KUKA KRL program: MyProgram_261().src

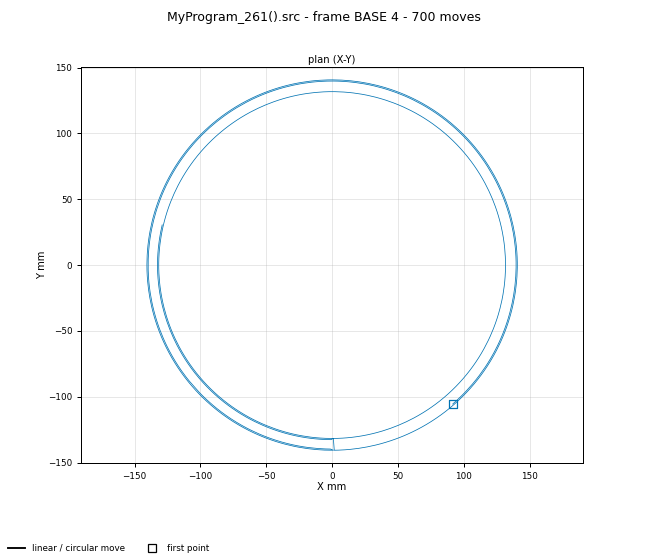
[picture p0: tool path of MyProgram_261().src in frame BASE 4, 700 of 700 moves have a stored position in this frame; points joined in program order, loops and branches not executed]
&ACCESS RVP
&REL 1
&PARAM TEMPLATE = C:\KRC\Roboter\Template\vorgabe
&PARAM EDITMASK = *
DEF MyProgram_261()
; ---- Setting reference (Base) ----
$BASE = BASE_DATA[4]

; --------------------------
; ---- Setting tool (TCP) ----
$TOOL = TOOL_DATA[3]
; --------------------------

$VEL.CP = VEL_APROX_PRINT
Startdeposition()
$VEL.CP = VEL_PRINT
LIN {X 91.5641,Y -105.5232,Z 167,A -46.4819,B 10.3454,C 0.2942,E1 10.4568,E2 497.4556} C_DIS
LIN {X 94.9436,Y -102.4931,Z 167,A -45.04,B 10.3452,C 0.3012,E1 10.4597,E2 496.067} C_DIS
LIN {X 98.56,Y -99.0198,Z 167,A -43.0358,B 10.3452,C 0.2981,E1 10.4637,E2 494.0674} C_DIS
LIN {X 101.6375,Y -95.8582,Z 167,A -40.8516,B 10.3456,C 0.2845,E1 10.468,E2 491.8321} C_DIS
LIN {X 104.5658,Y -92.6553,Z 167,A -39.6802,B 10.3453,C 0.2962,E1 10.47,E2 490.7387} C_DIS
LIN {X 106.6015,Y -90.306,Z 167,A -38.2518,B 10.3455,C 0.2893,E1 10.4727,E2 489.2889} C_DIS
LIN {X 109.2383,Y -87.0977,Z 167,A -36.5625,B 10.3456,C 0.2857,E1 10.4756,E2 487.5994} C_DIS
LIN {X 111.7975,Y -83.7884,Z 167,A -34.7726,B 10.3458,C 0.2796,E1 10.4787,E2 485.798} C_DIS
LIN {X 116.3977,Y -77.2703,Z 167,A -31.7918,B 10.3458,C 0.2792,E1 10.4834,E2 482.8518} C_DIS
LIN {X 118.3157,Y -74.3,Z 167,A -29.8592,B 10.3462,C 0.2629,E1 10.4864,E2 480.8544} C_DIS
LIN {X 120.3509,Y -70.9556,Z 167,A -28.8973,B 10.3459,C 0.2756,E1 10.4876,E2 479.975} C_DIS
LIN {X 122.8521,Y -66.5321,Z 167,A -26.472,B 10.3463,C 0.2612,E1 10.491,E2 477.5029} C_DIS
LIN {X 125.5362,Y -61.3138,Z 167,A -24.2471,B 10.3463,C 0.2596,E1 10.4938,E2 475.299} C_DIS
LIN {X 126.9956,Y -58.2302,Z 167,A -22.8435,B 10.3463,C 0.2557,E1 10.4954,E2 473.8932} C_DIS
LIN {X 128.5472,Y -54.7236,Z 167,A -21.1883,B 10.3465,C 0.2492,E1 10.4973,E2 472.2256} C_DIS
LIN {X 129.9617,Y -51.2729,Z 167,A -19.845,B 10.3465,C 0.2499,E1 10.4986,E2 470.9048} C_DIS
LIN {X 131.4593,Y -47.2962,Z 167,A -17.9921,B 10.3467,C 0.2421,E1 10.5004,E2 469.0356} C_DIS
LIN {X 132.6867,Y -43.7365,Z 167,A -16.549,B 10.3467,C 0.2405,E1 10.5017,E2 467.6039} C_DIS
LIN {X 133.7753,Y -40.2869,Z 167,A -14.9397,B 10.3469,C 0.233,E1 10.503,E2 465.9767} C_DIS
LIN {X 134.9483,Y -36.159,Z 167,A -12.8239,B 10.3472,C 0.2185,E1 10.5046,E2 463.8124} C_DIS
LIN {X 136.0946,Y -31.5754,Z 167,A -11.579,B 10.347,C 0.2313,E1 10.5054,E2 462.6559} C_DIS
LIN {X 136.6271,Y -29.183,Z 167,A -10.1588,B 10.3473,C 0.2174,E1 10.5062,E2 461.1805} C_DIS
LIN {X 137.2908,Y -25.8822,Z 167,A -9.1019,B 10.3472,C 0.222,E1 10.5068,E2 460.1643} C_DIS
LIN {X 137.8805,Y -22.5325,Z 167,A -7.7697,B 10.3472,C 0.2196,E1 10.5074,E2 458.8388} C_DIS
LIN {X 138.4173,Y -18.9686,Z 167,A -6.2808,B 10.3473,C 0.215,E1 10.508,E2 457.347} C_DIS
LIN {X 138.8085,Y -15.8511,Z 167,A -4.951,B 10.3474,C 0.2102,E1 10.5084,E2 456.0104} C_DIS
LIN {X 139.2347,Y -11.5036,Z 167,A -3.2691,B 10.3474,C 0.2078,E1 10.5089,E2 454.3408} C_DIS
LIN {X 139.4553,Y -8.4152,Z 167,A -1.8781,B 10.3476,C 0.2009,E1 10.5091,E2 452.9329} C_DIS
LIN {X 139.6307,Y -4.7299,Z 167,A -0.5083,B 10.3476,C 0.2003,E1 10.5093,E2 451.5801} C_DIS
LIN {X 139.698,Y -1.8215,Z 167,A 0.7879,B 10.3477,C 0.194,E1 10.5093,E2 450.2693} C_DIS
LIN {X 139.6853,Y 2.585,Z 167,A 2.554,B 10.3477,C 0.1898,E1 10.5093,E2 448.5067} C_DIS
LIN {X 139.5635,Y 6.4013,Z 167,A 4.1323,B 10.3479,C 0.1849,E1 10.5091,E2 446.9253} C_DIS
LIN {X 139.2836,Y 10.9175,Z 167,A 5.8225,B 10.3479,C 0.1839,E1 10.5088,E2 445.2548} C_DIS
LIN {X 138.9636,Y 14.4206,Z 167,A 7.4324,B 10.348,C 0.1753,E1 10.5083,E2 443.6218} C_DIS
LIN {X 138.2126,Y 20.4014,Z 167,A 9.8969,B 10.3482,C 0.1683,E1 10.5074,E2 441.156} C_DIS
LIN {X 137.4569,Y 24.9855,Z 167,A 11.6074,B 10.3482,C 0.168,E1 10.5066,E2 439.4689} C_DIS
LIN {X 136.0935,Y 31.5801,Z 167,A 14.2954,B 10.3482,C 0.1621,E1 10.505,E2 436.7881} C_DIS
LIN {X 135.3473,Y 34.6364,Z 167,A 15.6039,B 10.3483,C 0.1579,E1 10.5041,E2 435.4762} C_DIS
LIN {X 134.2036,Y 38.8338,Z 167,A 17.4103,B 10.3484,C 0.1524,E1 10.5028,E2 433.6654} C_DIS
LIN {X 133.11,Y 42.429,Z 167,A 18.9207,B 10.3484,C 0.1489,E1 10.5015,E2 432.1576} C_DIS
LIN {X 131.8259,Y 46.2676,Z 167,A 20.5108,B 10.3484,C 0.1462,E1 10.5001,E2 430.5753} C_DIS
LIN {X 130.1559,Y 50.7733,Z 167,A 23.2054,B 10.3488,C 0.1219,E1 10.4973,E2 427.7855} C_DIS
LIN {X 127.8483,Y 56.3369,Z 167,A 24.8587,B 10.3486,C 0.1367,E1 10.4956,E2 426.2361} C_DIS
LIN {X 125.7779,Y 60.8177,Z 167,A 26.8929,B 10.3486,C 0.1311,E1 10.4931,E2 424.1993} C_DIS
LIN {X 124.2977,Y 63.7865,Z 167,A 28.2687,B 10.3487,C 0.1272,E1 10.4914,E2 422.8205} C_DIS
LIN {X 122.3038,Y 67.5338,Z 167,A 31.1972,B 10.3491,C 0.0919,E1 10.4872,E2 419.737} C_DIS
LIN {X 117.8706,Y 75.0044,Z 167,A 33.3946,B 10.3488,C 0.1186,E1 10.4843,E2 417.7144} C_DIS
LIN {X 115.7064,Y 78.3008,Z 167,A 35.1536,B 10.3489,C 0.111,E1 10.4815,E2 415.9364} C_DIS
LIN {X 113.1061,Y 82.0122,Z 167,A 36.9886,B 10.3489,C 0.1073,E1 10.4785,E2 414.1033} C_DIS
LIN {X 110.2068,Y 85.8695,Z 167,A 38.8498,B 10.3489,C 0.1057,E1 10.4754,E2 412.2562} C_DIS
LIN {X 107.8694,Y 88.7882,Z 167,A 40.4684,B 10.349,C 0.1002,E1 10.4725,E2 410.626} C_DIS
LIN {X 105.0218,Y 92.1387,Z 167,A 42.5298,B 10.3491,C 0.0897,E1 10.4687,E2 408.5307} C_DIS
LIN {X 102.5085,Y 94.927,Z 167,A 43.6692,B 10.3491,C 0.0966,E1 10.4666,E2 407.4419} C_DIS
LIN {X 99.8331,Y 97.7361,Z 167,A 45.3434,B 10.3491,C 0.0912,E1 10.4633,E2 405.7564} C_DIS
LIN {X 96.8028,Y 100.739,Z 167,A 47.1278,B 10.3491,C 0.0868,E1 10.4598,E2 403.967} C_DIS
LIN {X 93.4543,Y 103.8527,Z 167,A 48.9847,B 10.3491,C 0.0836,E1 10.4559,E2 402.1117} C_DIS
LIN {X 89.4362,Y 107.3329,Z 167,A 51.0122,B 10.3491,C 0.0834,E1 10.4517,E2 400.103} C_DIS
LIN {X 86.3492,Y 109.8308,Z 167,A 52.694,B 10.3492,C 0.0791,E1 10.448,E2 398.414} C_DIS
LIN {X 82.9189,Y 112.4433,Z 167,A 54.4993,B 10.3492,C 0.0752,E1 10.4439,E2 396.6036} C_DIS
LIN {X 79.2864,Y 115.0336,Z 167,A 56.2762,B 10.3492,C 0.0735,E1 10.4399,E2 394.8331} C_DIS
LIN {X 75.6367,Y 117.4658,Z 167,A 58.0915,B 10.3492,C 0.0703,E1 10.4356,E2 393.0154} C_DIS
LIN {X 71.8064,Y 119.8455,Z 167,A 59.8903,B 10.3492,C 0.0688,E1 10.4314,E2 391.2228} C_DIS
LIN {X 68.0156,Y 122.037,Z 167,A 61.7048,B 10.3493,C 0.0658,E1 10.4269,E2 389.4057} C_DIS
LIN {X 64.1506,Y 124.1123,Z 167,A 63.3886,B 10.3493,C 0.0662,E1 10.4228,E2 387.7365} C_DIS
LIN {X 61.4926,Y 125.448,Z 167,A 64.6061,B 10.3493,C 0.0647,E1 10.4198,E2 386.5192} C_DIS
LIN {X 58.3333,Y 126.9479,Z 167,A 66.0262,B 10.3493,C 0.0633,E1 10.4162,E2 385.1009} C_DIS
LIN {X 54.9493,Y 128.4496,Z 167,A 67.6856,B 10.3493,C 0.0582,E1 10.4119,E2 383.4237} C_DIS
LIN {X 51.3398,Y 129.9356,Z 167,A 69.1204,B 10.3493,C 0.0605,E1 10.4082,E2 382.01} C_DIS
LIN {X 48.4623,Y 131.0351,Z 167,A 70.3602,B 10.3493,C 0.0599,E1 10.405,E2 380.7733} C_DIS
LIN {X 44.8622,Y 132.3119,Z 167,A 71.9098,B 10.3493,C 0.0588,E1 10.4009,E2 379.226} C_DIS
LIN {X 42.1564,Y 133.1971,Z 167,A 73.1116,B 10.3493,C 0.057,E1 10.3977,E2 378.02} C_DIS
LIN {X 38.2027,Y 134.3853,Z 167,A 75.716,B 10.3495,C 0.0341,E1 10.3904,E2 375.2998} C_DIS
LIN {X 31.6224,Y 136.0838,Z 167,A 77.5761,B 10.3494,C 0.0542,E1 10.3857,E2 373.5585} C_DIS
LIN {X 28.5214,Y 136.768,Z 167,A 79.3151,B 10.3494,C 0.0433,E1 10.3808,E2 371.7645} C_DIS
LIN {X 24.5396,Y 137.5367,Z 167,A 80.5343,B 10.3494,C 0.0528,E1 10.3776,E2 370.602} C_DIS
LIN {X 20.5345,Y 138.1936,Z 167,A 82.1615,B 10.3494,C 0.053,E1 10.3731,E2 368.9801} C_DIS
LIN {X 17.5042,Y 138.6094,Z 167,A 83.4751,B 10.3494,C 0.0512,E1 10.3694,E2 367.6594} C_DIS
LIN {X 12.4566,Y 139.1541,Z 167,A 85.4637,B 10.3494,C 0.0528,E1 10.3639,E2 365.6834} C_DIS
LIN {X 8.3518,Y 139.4592,Z 167,A 87.1865,B 10.3494,C 0.0518,E1 10.3591,E2 363.9568} C_DIS
LIN {X 4.5252,Y 139.6371,Z 167,A 88.7407,B 10.3494,C 0.052,E1 10.3548,E2 362.4054} C_DIS
LIN {X 1.0666,Y 139.7052,Z 167,A 90.2856,B 10.3494,C 0.0491,E1 10.3504,E2 360.8452} C_DIS
LIN {X -3.9161,Y 139.6541,Z 167,A 92.3097,B 10.3494,C 0.0498,E1 10.3448,E2 358.8246} C_DIS
LIN {X -8.5481,Y 139.4471,Z 167,A 94.2081,B 10.3494,C 0.0502,E1 10.3395,E2 356.9275} C_DIS
LIN {X -11.8169,Y 139.2082,Z 167,A 95.8533,B 10.3494,C 0.0438,E1 10.3348,E2 355.245} C_DIS
LIN {X -15.5616,Y 138.8404,Z 167,A 97.2474,B 10.3494,C 0.0477,E1 10.331,E2 353.8706} C_DIS
LIN {X -22.0151,Y 137.9647,Z 167,A 99.6967,B 10.3494,C 0.0539,E1 10.3243,E2 351.4509} C_DIS
LIN {X -25.2101,Y 137.4167,Z 167,A 101.3012,B 10.3494,C 0.0486,E1 10.3198,E2 349.8126} C_DIS
LIN {X -29.7519,Y 136.5043,Z 167,A 103.0354,B 10.3494,C 0.0534,E1 10.3152,E2 348.1006} C_DIS
LIN {X -33.502,Y 135.6345,Z 167,A 104.5307,B 10.3494,C 0.0564,E1 10.3111,E2 346.6168} C_DIS
LIN {X -36.4127,Y 134.8806,Z 167,A 105.779,B 10.3494,C 0.057,E1 10.3077,E2 345.3675} C_DIS
LIN {X -40.4129,Y 133.7368,Z 167,A 107.614,B 10.3494,C 0.0557,E1 10.3028,E2 343.5175} C_DIS
LIN {X -44.2758,Y 132.5071,Z 167,A 109.2421,B 10.3494,C 0.058,E1 10.2985,E2 341.8949} C_DIS
LIN {X -47.4884,Y 131.39,Z 167,A 110.6149,B 10.3494,C 0.0599,E1 10.2949,E2 340.526} C_DIS
LIN {X -50.9895,Y 130.0718,Z 167,A 112.0877,B 10.3494,C 0.0629,E1 10.2911,E2 339.0622} C_DIS
LIN {X -54.2261,Y 128.7562,Z 167,A 113.5626,B 10.3494,C 0.0637,E1 10.2873,E2 337.5831} C_DIS
LIN {X -57.3515,Y 127.3945,Z 167,A 114.9798,B 10.3494,C 0.065,E1 10.2836,E2 336.1647} C_DIS
LIN {X -61.0394,Y 125.6716,Z 167,A 117.1975,B 10.3494,C 0.0555,E1 10.2779,E2 333.8792} C_DIS
LIN {X -65.1846,Y 123.5697,Z 167,A 118.4147,B 10.3493,C 0.0728,E1 10.2751,E2 332.7505} C_DIS
LIN {X -70.0982,Y 120.8522,Z 167,A 120.7097,B 10.3493,C 0.0763,E1 10.2695,E2 330.4587} C_DIS
LIN {X -72.4715,Y 119.444,Z 167,A 122.1732,B 10.3493,C 0.0711,E1 10.2659,E2 328.9545} C_DIS
LIN {X -75.5503,Y 117.5211,Z 167,A 123.5269,B 10.3493,C 0.0763,E1 10.2628,E2 327.6192} C_DIS
LIN {X -78.6889,Y 115.4437,Z 167,A 125.1993,B 10.3493,C 0.0763,E1 10.2588,E2 325.932} C_DIS
LIN {X -82.3522,Y 112.8596,Z 167,A 127.065,B 10.3493,C 0.0789,E1 10.2546,E2 324.0647} C_DIS
LIN {X -86.4222,Y 109.7735,Z 167,A 129.0984,B 10.3492,C 0.084,E1 10.2501,E2 322.0411} C_DIS
LIN {X -89.8173,Y 107.0133,Z 167,A 130.9375,B 10.3492,C 0.0864,E1 10.2462,E2 320.1981} C_DIS
LIN {X -93.073,Y 104.1942,Z 167,A 132.7488,B 10.3492,C 0.089,E1 10.2424,E2 318.3829} C_DIS
LIN {X -96.5984,Y 100.9343,Z 167,A 134.6683,B 10.3491,C 0.094,E1 10.2385,E2 316.4717} C_DIS
LIN {X -99.3648,Y 98.2128,Z 167,A 136.2739,B 10.3491,C 0.0971,E1 10.2353,E2 314.866} C_DIS
LIN {X -102.3614,Y 95.085,Z 167,A 138.1179,B 10.3491,C 0.0996,E1 10.2318,E2 313.0152} C_DIS
LIN {X -105.5448,Y 91.5389,Z 167,A 140.8044,B 10.3491,C 0.0889,E1 10.2267,E2 310.2379} C_DIS
LIN {X -109.4122,Y 86.8791,Z 167,A 142.3815,B 10.3489,C 0.1132,E1 10.2241,E2 308.7784} C_DIS
LIN {X -111.4488,Y 84.2507,Z 167,A 144.3939,B 10.349,C 0.1032,E1 10.2206,E2 306.6854} C_DIS
LIN {X -114.0628,Y 80.6766,Z 167,A 145.6477,B 10.3488,C 0.119,E1 10.2187,E2 305.5047} C_DIS
LIN {X -116.056,Y 77.7821,Z 167,A 147.3134,B 10.3488,C 0.118,E1 10.216,E2 303.8124} C_DIS
LIN {X -118.4654,Y 74.0609,Z 167,A 149.1318,B 10.3488,C 0.1226,E1 10.2133,E2 301.9959} C_DIS
LIN {X -120.7426,Y 70.2875,Z 167,A 150.9547,B 10.3488,C 0.1268,E1 10.2107,E2 300.173} C_DIS
LIN {X -122.9148,Y 66.4158,Z 167,A 152.8253,B 10.3487,C 0.1306,E1 10.2082,E2 298.2981} C_DIS
LIN {X -125.8203,Y 60.728,Z 167,A 155.4007,B 10.3486,C 0.1384,E1 10.205,E2 295.7311} C_DIS
LIN {X -127.4918,Y 57.134,Z 167,A 157.0773,B 10.3486,C 0.1417,E1 10.203,E2 294.0498} C_DIS
LIN {X -129.0103,Y 53.6177,Z 167,A 158.6859,B 10.3486,C 0.1452,E1 10.2012,E2 292.4382} C_DIS
LIN {X -130.3496,Y 50.2749,Z 167,A 160.1865,B 10.3485,C 0.1488,E1 10.1997,E2 290.9362} C_DIS
LIN {X -131.7965,Y 46.3524,Z 167,A 161.9403,B 10.3484,C 0.1528,E1 10.1981,E2 289.1794} C_DIS
LIN {X -132.8123,Y 43.359,Z 167,A 163.1434,B 10.3484,C 0.1583,E1 10.197,E2 287.9896} C_DIS
LIN {X -133.7109,Y 40.4973,Z 167,A 164.4128,B 10.3483,C 0.161,E1 10.196,E2 286.7165} C_DIS
LIN {X -134.8267,Y 36.6149,Z 167,A 165.9985,B 10.3482,C 0.1671,E1 10.1948,E2 285.1416} C_DIS
LIN {X -135.5363,Y 33.8919,Z 167,A 167.2528,B 10.3482,C 0.1684,E1 10.1939,E2 283.8758} C_DIS
LIN {X -136.3106,Y 30.6295,Z 167,A 168.6191,B 10.3481,C 0.1725,E1 10.1931,E2 282.5121} C_DIS
LIN {X -136.9712,Y 27.523,Z 167,A 169.9577,B 10.3481,C 0.1755,E1 10.1923,E2 281.1703} C_DIS
LIN {X -137.6448,Y 23.9357,Z 167,A 171.631,B 10.3481,C 0.1764,E1 10.1915,E2 279.4762} C_DIS
LIN {X -138.2663,Y 20.0262,Z 167,A 173.227,B 10.3479,C 0.1816,E1 10.1908,E2 277.8854} C_DIS
LIN {X -138.8367,Y 15.5998,Z 167,A 175.5912,B 10.348,C 0.1764,E1 10.19,E2 275.455} C_DIS
LIN {X -139.3012,Y 10.6777,Z 167,A 176.9468,B 10.3477,C 0.1956,E1 10.1897,E2 274.1872} C_DIS
LIN {X -139.6441,Y 4.2731,Z 167,A 179.5436,B 10.3475,C 0.204,E1 10.1894,E2 271.5976} C_DIS
LIN {X -139.6627,Y -3.6064,Z 167,A -177.1518,B 10.3474,C 0.2121,E1 10.1894,E2 268.2871} C_DIS
LIN {X -139.3859,Y -9.5167,Z 167,A -174.6168,B 10.3473,C 0.217,E1 10.1898,E2 265.7408} C_DIS
LIN {X -139.0526,Y -13.5262,Z 167,A -172.8775,B 10.3472,C 0.22,E1 10.1902,E2 263.9917} C_DIS
LIN {X -138.6677,Y -17.0307,Z 167,A -171.2731,B 10.3472,C 0.2211,E1 10.1907,E2 262.3685} C_DIS
LIN {X -138.0837,Y -21.2471,Z 167,A -169.5831,B 10.347,C 0.2272,E1 10.1914,E2 260.6872} C_DIS
LIN {X -137.3847,Y -25.389,Z 167,A -167.8954,B 10.347,C 0.2328,E1 10.1922,E2 259.0055} C_DIS
LIN {X -136.7967,Y -28.3805,Z 167,A -166.627,B 10.3468,C 0.236,E1 10.1929,E2 257.7359} C_DIS
LIN {X -136.1454,Y -31.3526,Z 167,A -165.3428,B 10.3468,C 0.2388,E1 10.1937,E2 256.4481} C_DIS
LIN {X -135.2817,Y -34.8949,Z 167,A -163.7904,B 10.3468,C 0.2419,E1 10.1948,E2 254.8897} C_DIS
LIN {X -134.0554,Y -39.34,Z 167,A -161.8798,B 10.3466,C 0.2468,E1 10.1962,E2 252.9781} C_DIS
LIN {X -133.0262,Y -42.6911,Z 167,A -160.3546,B 10.3466,C 0.249,E1 10.1975,E2 251.443} C_DIS
LIN {X -131.8385,Y -46.2313,Z 167,A -158.8262,B 10.3464,C 0.2532,E1 10.1989,E2 249.9162} C_DIS
LIN {X -130.6226,Y -49.5636,Z 167,A -157.4706,B 10.3464,C 0.2592,E1 10.2002,E2 248.5745} C_DIS
LIN {X -129.3637,Y -52.7619,Z 167,A -155.9956,B 10.3462,C 0.2616,E1 10.2017,E2 247.0921} C_DIS
LIN {X -128.1147,Y -55.7239,Z 167,A -154.6431,B 10.3462,C 0.2644,E1 10.2032,E2 245.7361} C_DIS
LIN {X -126.6352,Y -59.0095,Z 167,A -153.1439,B 10.3461,C 0.2678,E1 10.205,E2 244.2353} C_DIS
LIN {X -125.1029,Y -62.1923,Z 167,A -151.6775,B 10.346,C 0.2712,E1 10.2068,E2 242.7676} C_DIS
LIN {X -123.499,Y -65.3192,Z 167,A -150.2157,B 10.346,C 0.2745,E1 10.2087,E2 241.3041} C_DIS
LIN {X -121.3846,Y -69.1721,Z 167,A -148.3274,B 10.3458,C 0.2772,E1 10.2113,E2 239.406} C_DIS
LIN {X -119.155,Y -72.9459,Z 167,A -146.4946,B 10.3458,C 0.2809,E1 10.2139,E2 237.5697} C_DIS
LIN {X -116.7178,Y -76.785,Z 167,A -144.6117,B 10.3456,C 0.285,E1 10.2168,E2 235.6856} C_DIS
LIN {X -114.2962,Y -80.3456,Z 167,A -142.8335,B 10.3456,C 0.2889,E1 10.2196,E2 233.9069} C_DIS
LIN {X -110.7764,Y -85.1333,Z 167,A -140.4257,B 10.3454,C 0.2951,E1 10.2236,E2 231.5041} C_DIS
LIN {X -108.4435,Y -88.0862,Z 167,A -138.7727,B 10.3454,C 0.2962,E1 10.2265,E2 229.8377} C_DIS
LIN {X -100.7412,Y -96.8005,Z 167,A -134.298,B 10.3448,C 0.3125,E1 10.2348,E2 225.4036} C_DIS
LIN {X -98.2946,Y -99.2835,Z 167,A -132.5248,B 10.345,C 0.3081,E1 10.2384,E2 223.5866} C_DIS
LIN {X -94.9183,Y -102.5167,Z 167,A -130.6026,B 10.3449,C 0.3117,E1 10.2423,E2 221.6644} C_DIS
LIN {X -90.5585,Y -106.3868,Z 167,A -128.2061,B 10.3447,C 0.316,E1 10.2473,E2 219.2679} C_DIS
LIN {X -87.2992,Y -109.0778,Z 167,A -126.4445,B 10.3447,C 0.3184,E1 10.2511,E2 217.5031} C_DIS
LIN {X -83.7648,Y -111.815,Z 167,A -124.5726,B 10.3446,C 0.3206,E1 10.2553,E2 215.6266} C_DIS
LIN {X -80.1113,Y -114.461,Z 167,A -122.7099,B 10.3446,C 0.3233,E1 10.2596,E2 213.7626} C_DIS
LIN {X -76.3544,Y -117.0004,Z 167,A -120.8263,B 10.3444,C 0.3256,E1 10.2639,E2 211.8762} C_DIS
LIN {X -72.4782,Y -119.4401,Z 167,A -118.9407,B 10.3444,C 0.3282,E1 10.2684,E2 209.9899} C_DIS
LIN {X -68.5476,Y -121.7383,Z 167,A -117.0809,B 10.3443,C 0.3308,E1 10.2729,E2 208.1312} C_DIS
LIN {X -64.6048,Y -123.8741,Z 167,A -115.3201,B 10.3442,C 0.3349,E1 10.2772,E2 206.3807} C_DIS
LIN {X -61.4508,Y -125.4686,Z 167,A -113.8258,B 10.3442,C 0.3356,E1 10.281,E2 204.8805} C_DIS
LIN {X -58.1353,Y -127.0395,Z 167,A -112.3799,B 10.344,C 0.3386,E1 10.2846,E2 203.4422} C_DIS
LIN {X -55.436,Y -128.2392,Z 167,A -111.0427,B 10.344,C 0.3371,E1 10.2881,E2 202.0887} C_DIS
LIN {X -51.9113,Y -129.7066,Z 167,A -109.537,B 10.344,C 0.34,E1 10.292,E2 200.5907} C_DIS
LIN {X -47.7872,Y -131.2822,Z 167,A -107.6997,B 10.344,C 0.341,E1 10.2968,E2 198.7498} C_DIS
LIN {X -43.9717,Y -132.6084,Z 167,A -106.0808,B 10.3439,C 0.3432,E1 10.3011,E2 197.1355} C_DIS
LIN {X -38.4516,Y -134.3154,Z 167,A -103.1562,B 10.3442,C 0.3323,E1 10.3091,E2 194.1379} C_DIS
LIN {X -33.9914,Y -135.511,Z 167,A -101.7982,B 10.3438,C 0.3457,E1 10.3126,E2 192.8497} C_DIS
LIN {X -29.7938,Y -136.4952,Z 167,A -99.9983,B 10.3438,C 0.3459,E1 10.3175,E2 191.0453} C_DIS
LIN {X -26.2856,Y -137.2137,Z 167,A -98.5184,B 10.3438,C 0.3463,E1 10.3215,E2 189.5635} C_DIS
LIN {X -21.9898,Y -137.9687,Z 167,A -96.6335,B 10.3438,C 0.3447,E1 10.3268,E2 187.6655} C_DIS
LIN {X -18.0061,Y -138.5437,Z 167,A -95.0719,B 10.3438,C 0.3472,E1 10.3311,E2 186.1149} C_DIS
LIN {X -13.9116,Y -139.0156,Z 167,A -93.4162,B 10.3438,C 0.3483,E1 10.3357,E2 184.4632} C_DIS
LIN {X -10.837,Y -139.2895,Z 167,A -92.2253,B 10.3436,C 0.3502,E1 10.3389,E2 183.2817} C_DIS
LIN {X -8.1116,Y -139.474,Z 167,A -91.0794,B 10.3436,C 0.3497,E1 10.3421,E2 182.1319} C_DIS
LIN {X -5.1092,Y -139.6159,Z 167,A -89.6863,B 10.3438,C 0.3459,E1 10.3461,E2 180.7172} C_DIS
LIN {X -1.2526,Y -139.7042,Z 167,A -88.2497,B 10.3437,C 0.3492,E1 10.3501,E2 179.299} C_DIS
LIN {X -1.2526,Y -139.7042,Z 167,A -88.2497,B 10.3437,C 0.3492,E1 10.3501,E2 179.299} C_DIS
Enddeposition()
LIN {X 0.9939,Y -140.6192,Z 167,A -87.7668,B 10.3432,C 0.3656,E1 10.3513,E2 178.9073} C_DIS
Startdeposition()
$VEL.CP = VEL_PRINT
LIN {X -2.344,Y -140.605,Z 167,A -89.2479,B 10.3432,C 0.3686,E1 10.3471,E2 180.4049} C_DIS
LIN {X -5.7191,Y -140.5083,Z 167,A -90.6137,B 10.3432,C 0.3684,E1 10.3433,E2 181.7701} C_DIS
LIN {X -9.0449,Y -140.3338,Z 167,A -91.9784,B 10.3432,C 0.3684,E1 10.3395,E2 183.1363} C_DIS
LIN {X -12.4568,Y -140.0723,Z 167,A -93.3816,B 10.3432,C 0.3685,E1 10.3355,E2 184.5412} C_DIS
LIN {X -15.89,Y -139.7245,Z 167,A -94.7918,B 10.3432,C 0.3684,E1 10.3316,E2 185.9525} C_DIS
LIN {X -19.0266,Y -139.3333,Z 167,A -96.2005,B 10.343,C 0.3708,E1 10.3277,E2 187.3774} C_DIS
LIN {X -22.3393,Y -138.8409,Z 167,A -97.4561,B 10.3431,C 0.3679,E1 10.3243,E2 188.6193} C_DIS
LIN {X -25.7376,Y -138.2506,Z 167,A -98.8614,B 10.3431,C 0.3674,E1 10.3204,E2 190.025} C_DIS
LIN {X -29.1206,Y -137.5772,Z 167,A -100.2705,B 10.3431,C 0.3668,E1 10.3165,E2 191.4349} C_DIS
LIN {X -32.4911,Y -136.82,Z 167,A -101.6751,B 10.3432,C 0.366,E1 10.3127,E2 192.8395} C_DIS
LIN {X -35.8248,Y -135.985,Z 167,A -103.0786,B 10.3432,C 0.3652,E1 10.3089,E2 194.2437} C_DIS
LIN {X -39.1419,Y -135.0674,Z 167,A -104.4855,B 10.3432,C 0.3643,E1 10.3051,E2 195.6514} C_DIS
LIN {X -42.4423,Y -134.0668,Z 167,A -105.9828,B 10.3432,C 0.3654,E1 10.3011,E2 197.1609} C_DIS
LIN {X -46.3803,Y -132.7558,Z 167,A -107.5946,B 10.3433,C 0.3622,E1 10.2969,E2 198.7627} C_DIS
LIN {X -49.64,Y -131.5717,Z 167,A -109.0153,B 10.3433,C 0.3611,E1 10.2931,E2 200.1844} C_DIS
LIN {X -52.8828,Y -130.3021,Z 167,A -110.4423,B 10.3434,C 0.3599,E1 10.2894,E2 201.6126} C_DIS
LIN {X -56.6277,Y -128.7196,Z 167,A -112.1792,B 10.3434,C 0.3599,E1 10.285,E2 203.3601} C_DIS
LIN {X -60.1216,Y -127.1251,Z 167,A -113.745,B 10.3434,C 0.3582,E1 10.281,E2 204.926} C_DIS
LIN {X -63.2287,Y -125.609,Z 167,A -115.0863,B 10.3436,C 0.3551,E1 10.2777,E2 206.2585} C_DIS
LIN {X -66.8779,Y -123.7058,Z 167,A -116.8606,B 10.3436,C 0.3551,E1 10.2732,E2 208.0454} C_DIS
LIN {X -70.8108,Y -121.4976,Z 167,A -118.7639,B 10.3436,C 0.354,E1 10.2686,E2 209.957} C_DIS
LIN {X -74.7682,Y -119.1029,Z 167,A -120.6371,B 10.3437,C 0.3511,E1 10.2642,E2 211.8285} C_DIS
LIN {X -78.5492,Y -116.6439,Z 167,A -122.4827,B 10.3438,C 0.3485,E1 10.2599,E2 213.6749} C_DIS
LIN {X -82.2073,Y -114.0954,Z 167,A -124.2578,B 10.3439,C 0.3447,E1 10.2558,E2 215.4443} C_DIS
LIN {X -85.307,Y -111.7962,Z 167,A -125.9064,B 10.3439,C 0.3437,E1 10.2521,E2 217.1023} C_DIS
LIN {X -88.5435,Y -109.2511,Z 167,A -127.5455,B 10.3441,C 0.34,E1 10.2486,E2 218.736} C_DIS
LIN {X -91.8509,Y -106.4851,Z 167,A -129.3522,B 10.3441,C 0.3379,E1 10.2447,E2 220.5487} C_DIS
LIN {X -95.0762,Y -103.6155,Z 167,A -131.1467,B 10.3442,C 0.3353,E1 10.241,E2 222.3471} C_DIS
LIN {X -98.2099,Y -100.6508,Z 167,A -132.8533,B 10.3444,C 0.3309,E1 10.2376,E2 224.0466} C_DIS
LIN {X -101.2511,Y -97.5908,Z 167,A -134.4535,B 10.3446,C 0.324,E1 10.2345,E2 225.6258} C_DIS
LIN {X -103.6127,Y -95.0793,Z 167,A -136.0952,B 10.3446,C 0.3261,E1 10.2313,E2 227.2974} C_DIS
LIN {X -106.6086,Y -91.7075,Z 167,A -137.9402,B 10.3446,C 0.3223,E1 10.2279,E2 229.1425} C_DIS
LIN {X -109.251,Y -88.5437,Z 167,A -139.6184,B 10.3448,C 0.3186,E1 10.2249,E2 230.8198} C_DIS
LIN {X -111.9145,Y -85.1524,Z 167,A -141.3878,B 10.3448,C 0.3149,E1 10.2219,E2 232.5899} C_DIS
LIN {X -114.4747,Y -81.6776,Z 167,A -143.2015,B 10.345,C 0.312,E1 10.2189,E2 234.4097} C_DIS
LIN {X -116.9258,Y -78.1282,Z 167,A -144.9701,B 10.345,C 0.3081,E1 10.2161,E2 236.1788} C_DIS
LIN {X -119.3405,Y -74.3875,Z 167,A -146.8109,B 10.3452,C 0.3043,E1 10.2134,E2 238.0219} C_DIS
LIN {X -121.4979,Y -70.8103,Z 167,A -148.5855,B 10.3452,C 0.3016,E1 10.2108,E2 239.8048} C_DIS
LIN {X -123.7059,Y -66.8778,Z 167,A -150.4805,B 10.3454,C 0.2981,E1 10.2083,E2 241.7059} C_DIS
LIN {X -125.9075,Y -62.6308,Z 167,A -152.335,B 10.3456,C 0.2912,E1 10.2059,E2 243.5469} C_DIS
LIN {X -127.4886,Y -59.3455,Z 167,A -153.7897,B 10.3456,C 0.2867,E1 10.2042,E2 244.9967} C_DIS
LIN {X -128.9461,Y -56.108,Z 167,A -155.2635,B 10.3458,C 0.2835,E1 10.2025,E2 246.4729} C_DIS
LIN {X -130.3021,Y -52.8828,Z 167,A -156.7059,B 10.3458,C 0.28,E1 10.201,E2 247.9164} C_DIS
LIN {X -131.5717,Y -49.64,Z 167,A -158.1428,B 10.346,C 0.2765,E1 10.1995,E2 249.3544} C_DIS
LIN {X -132.7558,Y -46.3803,Z 167,A -159.6344,B 10.346,C 0.2743,E1 10.1981,E2 250.855} C_DIS
LIN {X -134.0578,Y -42.4708,Z 167,A -161.3335,B 10.3461,C 0.27,E1 10.1967,E2 252.5554} C_DIS
LIN {X -135.1369,Y -38.9046,Z 167,A -162.8494,B 10.3462,C 0.2658,E1 10.1955,E2 254.0697} C_DIS
LIN {X -136.1948,Y -35.017,Z 167,A -164.5066,B 10.3464,C 0.2615,E1 10.1943,E2 255.7274} C_DIS
LIN {X -137.0439,Y -31.5309,Z 167,A -165.9583,B 10.3464,C 0.2572,E1 10.1934,E2 257.1766} C_DIS
LIN {X -137.7649,Y -28.2141,Z 167,A -167.3593,B 10.3465,C 0.2536,E1 10.1925,E2 258.5787} C_DIS
LIN {X -138.4019,Y -24.9023,Z 167,A -168.7487,B 10.3466,C 0.25,E1 10.1918,E2 259.9688} C_DIS
LIN {X -138.9011,Y -21.9514,Z 167,A -170.0027,B 10.3466,C 0.2472,E1 10.1913,E2 261.2261} C_DIS
LIN {X -139.3976,Y -18.5358,Z 167,A -171.3162,B 10.3468,C 0.2413,E1 10.1908,E2 262.5265} C_DIS
LIN {X -139.7683,Y -15.4996,Z 167,A -172.6958,B 10.3468,C 0.2403,E1 10.1903,E2 263.9219} C_DIS
LIN {X -140.106,Y -12.0655,Z 167,A -174.1224,B 10.3469,C 0.2366,E1 10.1899,E2 265.3498} C_DIS
LIN {X -140.3998,Y -7.9453,Z 167,A -175.9254,B 10.347,C 0.2341,E1 10.1896,E2 267.1663} C_DIS
LIN {X -140.5664,Y -4.0448,Z 167,A -177.4683,B 10.3471,C 0.2285,E1 10.1895,E2 268.7016} C_DIS
LIN {X -140.6258,Y 0.1845,Z 167,A -179.2531,B 10.3472,C 0.2247,E1 10.1895,E2 270.4926} C_DIS
LIN {X -140.5664,Y 4.0448,Z 167,A 179.2326,B 10.3473,C 0.2189,E1 10.1895,E2 271.9978} C_DIS
LIN {X -140.4309,Y 7.3822,Z 167,A 177.8557,B 10.3474,C 0.2153,E1 10.1897,E2 273.3753} C_DIS
LIN {X -140.2147,Y 10.7366,Z 167,A 176.355,B 10.3474,C 0.2138,E1 10.19,E2 274.8912} C_DIS
LIN {X -139.8369,Y 14.8622,Z 167,A 174.7203,B 10.3476,C 0.2079,E1 10.1904,E2 276.5174} C_DIS
LIN {X -139.3975,Y 18.5367,Z 167,A 173.172,B 10.3476,C 0.2043,E1 10.191,E2 278.0693} C_DIS
LIN {X -138.8408,Y 22.34,Z 167,A 171.6066,B 10.3477,C 0.1997,E1 10.1916,E2 279.6331} C_DIS
LIN {X -138.2499,Y 25.7408,Z 167,A 170.1746,B 10.3477,C 0.1962,E1 10.1924,E2 281.0667} C_DIS
LIN {X -137.5582,Y 29.2085,Z 167,A 168.7493,B 10.3479,C 0.1917,E1 10.1931,E2 282.4885} C_DIS
LIN {X -136.8198,Y 32.4922,Z 167,A 167.3336,B 10.3479,C 0.1886,E1 10.194,E2 283.9083} C_DIS
LIN {X -135.9802,Y 35.8429,Z 167,A 165.9089,B 10.3479,C 0.185,E1 10.195,E2 285.3337} C_DIS
LIN {X -135.0599,Y 39.1675,Z 167,A 164.4844,B 10.348,C 0.1814,E1 10.1961,E2 286.7591} C_DIS
LIN {X -134.0585,Y 42.4683,Z 167,A 162.9781,B 10.348,C 0.1794,E1 10.1974,E2 288.2765} C_DIS
LIN {X -132.7558,Y 46.3803,Z 167,A 161.3551,B 10.3482,C 0.1736,E1 10.1988,E2 289.8904} C_DIS
LIN {X -131.5717,Y 49.64,Z 167,A 159.9212,B 10.3482,C 0.1701,E1 10.2002,E2 291.3255} C_DIS
LIN {X -130.3021,Y 52.8828,Z 167,A 158.4812,B 10.3482,C 0.1666,E1 10.2017,E2 292.7665} C_DIS
LIN {X -128.7186,Y 56.6299,Z 167,A 156.6928,B 10.3483,C 0.1647,E1 10.2037,E2 294.5697} C_DIS
LIN {X -127.1437,Y 60.0826,Z 167,A 155.187,B 10.3483,C 0.1598,E1 10.2055,E2 296.0687} C_DIS
LIN {X -125.6235,Y 63.2002,Z 167,A 153.804,B 10.3485,C 0.1554,E1 10.2072,E2 297.4463} C_DIS
LIN {X -123.7059,Y 66.8779,Z 167,A 152.0143,B 10.3485,C 0.153,E1 10.2095,E2 299.2468} C_DIS
LIN {X -121.4977,Y 70.8105,Z 167,A 150.0992,B 10.3485,C 0.1498,E1 10.2122,E2 301.1696} C_DIS
LIN {X -119.1029,Y 74.7682,Z 167,A 148.2154,B 10.3486,C 0.1451,E1 10.2149,E2 303.0512} C_DIS
LIN {X -116.6439,Y 78.5492,Z 167,A 146.3895,B 10.3486,C 0.1403,E1 10.2178,E2 304.8736} C_DIS
LIN {X -114.2009,Y 82.0604,Z 167,A 144.6247,B 10.3487,C 0.1365,E1 10.2206,E2 306.6393} C_DIS
LIN {X -111.6014,Y 85.5617,Z 167,A 142.8495,B 10.3487,C 0.1323,E1 10.2236,E2 308.4124} C_DIS
LIN {X -108.8311,Y 89.0587,Z 167,A 141.0033,B 10.3488,C 0.1286,E1 10.2268,E2 310.2602} C_DIS
LIN {X -106.0488,Y 92.3543,Z 167,A 139.19,B 10.3488,C 0.1258,E1 10.2301,E2 312.0787} C_DIS
LIN {X -103.0102,Y 95.7318,Z 167,A 137.3072,B 10.3489,C 0.1224,E1 10.2337,E2 313.9636} C_DIS
LIN {X -99.7677,Y 99.1063,Z 167,A 135.4131,B 10.3489,C 0.1181,E1 10.2374,E2 315.8541} C_DIS
LIN {X -96.7644,Y 102.0414,Z 167,A 133.6431,B 10.3489,C 0.1157,E1 10.2409,E2 317.6297} C_DIS
LIN {X -93.367,Y 105.1586,Z 167,A 131.7666,B 10.349,C 0.1119,E1 10.2448,E2 319.5041} C_DIS
LIN {X -90.0109,Y 108.0457,Z 167,A 130.0029,B 10.349,C 0.1076,E1 10.2486,E2 321.261} C_DIS
LIN {X -87.0428,Y 110.4503,Z 167,A 128.353,B 10.349,C 0.1067,E1 10.2522,E2 322.921} C_DIS
LIN {X -83.5485,Y 113.1169,Z 167,A 126.5467,B 10.3491,C 0.1038,E1 10.2562,E2 324.7275} C_DIS
LIN {X -79.8503,Y 115.7571,Z 167,A 124.7209,B 10.3491,C 0.1001,E1 10.2604,E2 326.5483} C_DIS
LIN {X -76.3017,Y 118.1262,Z 167,A 122.9653,B 10.3491,C 0.0976,E1 10.2645,E2 328.3045} C_DIS
LIN {X -72.8662,Y 120.2755,Z 167,A 121.2689,B 10.3491,C 0.0959,E1 10.2685,E2 330.005} C_DIS
LIN {X -68.7356,Y 122.683,Z 167,A 119.3522,B 10.3492,C 0.0923,E1 10.2731,E2 331.9161} C_DIS
LIN {X -64.5476,Y 124.9376,Z 167,A 117.3498,B 10.3492,C 0.091,E1 10.2781,E2 333.9249} C_DIS
LIN {X -60.9038,Y 126.7514,Z 167,A 115.7978,B 10.3492,C 0.0865,E1 10.282,E2 335.4621} C_DIS
LIN {X -57.7755,Y 128.2078,Z 167,A 114.3575,B 10.3492,C 0.0855,E1 10.2856,E2 336.9055} C_DIS
LIN {X -54.4963,Y 129.6355,Z 167,A 112.9111,B 10.3492,C 0.0835,E1 10.2893,E2 338.3494} C_DIS
LIN {X -51.264,Y 130.9475,Z 167,A 111.4824,B 10.3492,C 0.0821,E1 10.293,E2 339.7778} C_DIS
LIN {X -48.0132,Y 132.174,Z 167,A 110.0604,B 10.3493,C 0.0807,E1 10.2968,E2 341.1996} C_DIS
LIN {X -44.4856,Y 133.4023,Z 167,A 108.471,B 10.3493,C 0.0807,E1 10.301,E2 342.7962} C_DIS
LIN {X -40.4443,Y 134.6836,Z 167,A 106.8334,B 10.3493,C 0.0772,E1 10.3053,E2 344.4214} C_DIS
LIN {X -37.1282,Y 135.6352,Z 167,A 105.3854,B 10.3493,C 0.0769,E1 10.3092,E2 345.8737} C_DIS
LIN {X -33.7907,Y 136.505,Z 167,A 103.9755,B 10.3493,C 0.076,E1 10.313,E2 347.2832} C_DIS
LIN {X -30.4322,Y 137.2928,Z 167,A 102.5648,B 10.3493,C 0.0751,E1 10.3169,E2 348.6936} C_DIS
LIN {X -27.0532,Y 137.9984,Z 167,A 101.1528,B 10.3493,C 0.0743,E1 10.3207,E2 350.1054} C_DIS
LIN {X -23.6542,Y 138.6214,Z 167,A 99.739,B 10.3493,C 0.0737,E1 10.3246,E2 351.519} C_DIS
LIN {X -20.2484,Y 139.1594,Z 167,A 98.329,B 10.3493,C 0.0731,E1 10.3285,E2 352.9289} C_DIS
LIN {X -17.2313,Y 139.5659,Z 167,A 97.0804,B 10.3493,C 0.0728,E1 10.332,E2 354.1777} C_DIS
LIN {X -13.8072,Y 139.9454,Z 167,A 95.6723,B 10.3493,C 0.0724,E1 10.3359,E2 355.5857} C_DIS
LIN {X -9.8812,Y 140.2773,Z 167,A 94.0955,B 10.3493,C 0.0714,E1 10.3403,E2 357.158} C_DIS
LIN {X -6.5688,Y 140.4718,Z 167,A 92.7066,B 10.3493,C 0.0719,E1 10.3441,E2 358.5508} C_DIS
LIN {X -3.2681,Y 140.588,Z 167,A 91.404,B 10.3493,C 0.0708,E1 10.3478,E2 359.8474} C_DIS
LIN {X 0.4526,Y 140.6242,Z 167,A 89.8206,B 10.3493,C 0.0722,E1 10.3522,E2 361.4385} C_DIS
LIN {X 4.0448,Y 140.5664,Z 167,A 88.4096,B 10.3493,C 0.0711,E1 10.3561,E2 362.8423} C_DIS
LIN {X 7.3822,Y 140.4309,Z 167,A 87.0532,B 10.3493,C 0.0711,E1 10.3599,E2 364.1975} C_DIS
LIN {X 10.7367,Y 140.2146,Z 167,A 85.6685,B 10.3493,C 0.0717,E1 10.3638,E2 365.5836} C_DIS
LIN {X 14.174,Y 139.909,Z 167,A 84.2643,B 10.3493,C 0.072,E1 10.3677,E2 366.9871} C_DIS
LIN {X 17.6524,Y 139.5126,Z 167,A 82.9535,B 10.3493,C 0.0697,E1 10.3713,E2 368.2829} C_DIS
LIN {X 20.6953,Y 139.0955,Z 167,A 81.6027,B 10.3493,C 0.0725,E1 10.375,E2 369.6458} C_DIS
LIN {X 24.0392,Y 138.5563,Z 167,A 80.2038,B 10.3493,C 0.0736,E1 10.3789,E2 371.0467} C_DIS
LIN {X 27.4293,Y 137.9246,Z 167,A 78.7903,B 10.3493,C 0.0745,E1 10.3828,E2 372.4608} C_DIS
LIN {X 30.7908,Y 137.2129,Z 167,A 77.4156,B 10.3493,C 0.0747,E1 10.3865,E2 373.832} C_DIS
LIN {X 34.126,Y 136.4214,Z 167,A 76.0214,B 10.3493,C 0.0755,E1 10.3903,E2 375.2256} C_DIS
LIN {X 37.4611,Y 135.5433,Z 167,A 74.6099,B 10.3493,C 0.0767,E1 10.3941,E2 376.6376} C_DIS
LIN {X 40.8218,Y 134.5691,Z 167,A 73.2028,B 10.3493,C 0.0774,E1 10.3979,E2 378.0422} C_DIS
LIN {X 44.4847,Y 133.4026,Z 167,A 71.6036,B 10.3493,C 0.0795,E1 10.4021,E2 379.6453} C_DIS
LIN {X 48.0132,Y 132.174,Z 167,A 70.0659,B 10.3493,C 0.0813,E1 10.4062,E2 381.1848} C_DIS
LIN {X 52.2141,Y 130.5716,Z 167,A 68.2221,B 10.3493,C 0.0835,E1 10.411,E2 383.03} C_DIS
LIN {X 55.4015,Y 129.2516,Z 167,A 66.9108,B 10.3493,C 0.0828,E1 10.4143,E2 384.3293} C_DIS
LIN {X 58.7342,Y 127.7712,Z 167,A 65.4872,B 10.3493,C 0.083,E1 10.4179,E2 385.745} C_DIS
LIN {X 61.8585,Y 126.2885,Z 167,A 64.0948,B 10.3493,C 0.0843,E1 10.4214,E2 387.1354} C_DIS
LIN {X 65.042,Y 124.6786,Z 167,A 62.5729,B 10.3493,C 0.0879,E1 10.4252,E2 388.666} C_DIS
LIN {X 68.7336,Y 122.6841,Z 167,A 60.7778,B 10.3493,C 0.0923,E1 10.4296,E2 390.472} C_DIS
LIN {X 72.8666,Y 120.2752,Z 167,A 58.8696,B 10.3492,C 0.0941,E1 10.4342,E2 392.3754} C_DIS
LIN {X 76.736,Y 117.8443,Z 167,A 57.03,B 10.3492,C 0.0964,E1 10.4385,E2 394.2124} C_DIS
LIN {X 80.2673,Y 115.4678,Z 167,A 55.3082,B 10.3492,C 0.0989,E1 10.4425,E2 395.933} C_DIS
LIN {X 83.6436,Y 113.0468,Z 167,A 53.6278,B 10.3492,C 0.1015,E1 10.4463,E2 397.6122} C_DIS
LIN {X 87.1963,Y 110.3296,Z 167,A 51.8911,B 10.3492,C 0.1026,E1 10.4501,E2 399.3385} C_DIS
LIN {X 90.1208,Y 107.9538,Z 167,A 50.27,B 10.3491,C 0.1075,E1 10.4536,E2 400.9708} C_DIS
LIN {X 93.5607,Y 104.9865,Z 167,A 48.4764,B 10.3491,C 0.1096,E1 10.4574,E2 402.7577} C_DIS
LIN {X 96.7644,Y 102.0414,Z 167,A 46.7361,B 10.3491,C 0.1122,E1 10.4609,E2 404.4946} C_DIS
LIN {X 99.5764,Y 99.2988,Z 167,A 45.085,B 10.349,C 0.1167,E1 10.4642,E2 406.1526} C_DIS
LIN {X 102.6814,Y 96.0849,Z 167,A 43.2701,B 10.349,C 0.1204,E1 10.4677,E2 407.9675} C_DIS
LIN {X 105.8249,Y 92.6109,Z 167,A 41.4036,B 10.3489,C 0.1234,E1 10.4712,E2 409.8295} C_DIS
LIN {X 108.7057,Y 89.2121,Z 167,A 39.5957,B 10.3489,C 0.1272,E1 10.4744,E2 411.6373} C_DIS
LIN {X 111.3907,Y 85.8366,Z 167,A 37.9418,B 10.3489,C 0.1286,E1 10.4772,E2 413.2789} C_DIS
LIN {X 113.9714,Y 82.3785,Z 167,A 36.1604,B 10.3488,C 0.1333,E1 10.4802,E2 415.0643} C_DIS
LIN {X 116.4442,Y 78.8441,Z 167,A 34.4015,B 10.3488,C 0.1375,E1 10.483,E2 416.8244} C_DIS
LIN {X 118.9125,Y 75.0697,Z 167,A 32.6054,B 10.3487,C 0.1409,E1 10.4857,E2 418.6162} C_DIS
LIN {X 121.0588,Y 71.5582,Z 167,A 30.9861,B 10.3487,C 0.1436,E1 10.488,E2 420.2293} C_DIS
LIN {X 123.1987,Y 67.8076,Z 167,A 29.2874,B 10.3486,C 0.1465,E1 10.4903,E2 421.9213} C_DIS
LIN {X 124.9829,Y 64.4586,Z 167,A 27.6784,B 10.3486,C 0.152,E1 10.4924,E2 423.5394} C_DIS
LIN {X 126.7507,Y 60.9052,Z 167,A 26.1696,B 10.3485,C 0.1534,E1 10.4943,E2 425.0354} C_DIS
LIN {X 128.2077,Y 57.7758,Z 167,A 24.7573,B 10.3485,C 0.1573,E1 10.4959,E2 426.4494} C_DIS
LIN {X 129.6355,Y 54.4963,Z 167,A 23.338,B 10.3484,C 0.1602,E1 10.4975,E2 427.865} C_DIS
LIN {X 130.9475,Y 51.264,Z 167,A 21.9359,B 10.3484,C 0.1635,E1 10.4989,E2 429.2657} C_DIS
LIN {X 132.174,Y 48.0132,Z 167,A 20.54,B 10.3483,C 0.1669,E1 10.5003,E2 430.6602} C_DIS
LIN {X 133.4027,Y 44.4842,Z 167,A 18.9789,B 10.3483,C 0.1721,E1 10.5017,E2 432.2275} C_DIS
LIN {X 134.6836,Y 40.4446,Z 167,A 17.2161,B 10.3481,C 0.1778,E1 10.5031,E2 433.9963} C_DIS
LIN {X 135.8034,Y 36.5059,Z 167,A 15.692,B 10.3481,C 0.1787,E1 10.5043,E2 435.5033} C_DIS
LIN {X 136.6512,Y 33.1914,Z 167,A 14.3181,B 10.3481,C 0.1821,E1 10.5052,E2 436.8759} C_DIS
LIN {X 137.415,Y 29.872,Z 167,A 12.9514,B 10.348,C 0.1855,E1 10.506,E2 438.241} C_DIS
LIN {X 138.0944,Y 26.5545,Z 167,A 11.5938,B 10.348,C 0.1889,E1 10.5068,E2 439.597} C_DIS
LIN {X 138.6882,Y 23.2546,Z 167,A 10.3361,B 10.3479,C 0.19,E1 10.5074,E2 440.842} C_DIS
LIN {X 139.1596,Y 20.2469,Z 167,A 9.0107,B 10.3478,C 0.1958,E1 10.5079,E2 442.1795} C_DIS
LIN {X 139.5669,Y 17.2229,Z 167,A 7.7765,B 10.3478,C 0.1991,E1 10.5083,E2 443.4137} C_DIS
LIN {X 139.9478,Y 13.7826,Z 167,A 6.3936,B 10.3477,C 0.2025,E1 10.5088,E2 444.7945} C_DIS
LIN {X 140.2773,Y 9.8812,Z 167,A 4.8447,B 10.3476,C 0.206,E1 10.5091,E2 446.3389} C_DIS
LIN {X 140.5023,Y 5.8608,Z 167,A 3.1972,B 10.3475,C 0.2109,E1 10.5093,E2 447.9888} C_DIS
LIN {X 140.6087,Y 2.1188,Z 167,A 1.6826,B 10.3475,C 0.2151,E1 10.5094,E2 449.5036} C_DIS
LIN {X 140.6087,Y -2.1184,Z 167,A -0.0351,B 10.3473,C 0.2199,E1 10.5094,E2 451.2219} C_DIS
LIN {X 140.5083,Y -5.7191,Z 167,A -1.4274,B 10.3473,C 0.2223,E1 10.5093,E2 452.606} C_DIS
LIN {X 140.3338,Y -9.0449,Z 167,A -2.7722,B 10.3472,C 0.2259,E1 10.509,E2 453.9507} C_DIS
LIN {X 140.019,Y -13.0346,Z 167,A -4.4042,B 10.3471,C 0.2307,E1 10.5087,E2 455.5844} C_DIS
LIN {X 139.6501,Y -16.525,Z 167,A -5.7888,B 10.3471,C 0.2337,E1 10.5082,E2 456.9647} C_DIS
LIN {X 139.2199,Y -19.8246,Z 167,A -7.1132,B 10.3469,C 0.2368,E1 10.5077,E2 458.2865} C_DIS
LIN {X 138.5562,Y -24.0398,Z 167,A -8.8585,B 10.3469,C 0.2421,E1 10.5069,E2 460.0346} C_DIS
LIN {X 137.9244,Y -27.4304,Z 167,A -10.3276,B 10.3467,C 0.2478,E1 10.5062,E2 461.5134} C_DIS
LIN {X 137.2116,Y -30.7965,Z 167,A -11.6169,B 10.3467,C 0.2489,E1 10.5054,E2 462.7897} C_DIS
LIN {X 136.4203,Y -34.1303,Z 167,A -13.0073,B 10.3466,C 0.2527,E1 10.5045,E2 464.1808} C_DIS
LIN {X 135.5304,Y -37.5075,Z 167,A -14.3981,B 10.3465,C 0.256,E1 10.5035,E2 465.5691} C_DIS
LIN {X 134.5691,Y -40.822,Z 167,A -15.7839,B 10.3465,C 0.2594,E1 10.5024,E2 466.9537} C_DIS
LIN {X 133.4025,Y -44.4849,Z 167,A -17.3679,B 10.3463,C 0.2643,E1 10.501,E2 468.5417} C_DIS
LIN {X 132.174,Y -48.0132,Z 167,A -18.8315,B 10.3463,C 0.267,E1 10.4996,E2 469.9994} C_DIS
LIN {X 130.9475,Y -51.264,Z 167,A -20.2297,B 10.3461,C 0.2705,E1 10.4982,E2 471.397} C_DIS
LIN {X 129.6355,Y -54.4963,Z 167,A -21.718,B 10.346,C 0.2761,E1 10.4966,E2 472.8956} C_DIS
LIN {X 127.8529,Y -58.5577,Z 167,A -23.4318,B 10.346,C 0.2786,E1 10.4947,E2 474.5992} C_DIS
LIN {X 126.2915,Y -61.8524,Z 167,A -24.814,B 10.3459,C 0.2799,E1 10.493,E2 475.9696} C_DIS
LIN {X 124.8247,Y -64.7639,Z 167,A -26.2907,B 10.3457,C 0.2873,E1 10.4911,E2 477.4671} C_DIS
LIN {X 122.6841,Y -68.7336,Z 167,A -28.1121,B 10.3456,C 0.2917,E1 10.4887,E2 479.2885} C_DIS
LIN {X 120.2743,Y -72.8682,Z 167,A -30.0106,B 10.3454,C 0.2953,E1 10.486,E2 481.1824} C_DIS
LIN {X 117.8767,Y -76.686,Z 167,A -31.8261,B 10.3454,C 0.2994,E1 10.4833,E2 482.9972} C_DIS
LIN {X 115.4708,Y -80.263,Z 167,A -33.5544,B 10.3452,C 0.3031,E1 10.4805,E2 484.7238} C_DIS
LIN {X 112.9517,Y -83.7714,Z 167,A -35.2565,B 10.3452,C 0.3059,E1 10.4777,E2 486.4203} C_DIS
LIN {X 110.3296,Y -87.1964,Z 167,A -36.9614,B 10.3451,C 0.3087,E1 10.4748,E2 488.1203} C_DIS
LIN {X 107.9538,Y -90.1208,Z 167,A -38.5781,B 10.3449,C 0.3144,E1 10.4719,E2 489.7493} C_DIS
LIN {X 104.9865,Y -93.5607,Z 167,A -40.3654,B 10.3449,C 0.3169,E1 10.4687,E2 491.5302} C_DIS
LIN {X 102.0414,Y -96.7644,Z 167,A -42.1066,B 10.3447,C 0.3201,E1 10.4654,E2 493.2692} C_DIS
LIN {X 99.2989,Y -99.5764,Z 167,A -43.7566,B 10.3446,C 0.3248,E1 10.4621,E2 494.9274} C_DIS
LIN {X 96.0849,Y -102.6814,Z 167,A -45.5712,B 10.3445,C 0.3285,E1 10.4584,E2 496.7431} C_DIS
LIN {X 92.7279,Y -105.7228,Z 167,A -47.3674,B 10.3444,C 0.331,E1 10.4547,E2 498.5347} C_DIS
LIN {X 89.3261,Y -108.6126,Z 167,A -49.1014,B 10.3444,C 0.3324,E1 10.451,E2 500.2595} C_DIS
LIN {X 85.9917,Y -111.2705,Z 167,A -50.852,B 10.3442,C 0.336,E1 10.4471,E2 502.0136} C_DIS
LIN {X 82.8033,Y -113.6634,Z 167,A -52.5323,B 10.3441,C 0.3404,E1 10.4433,E2 503.7028} C_DIS
LIN {X 79.0064,Y -116.3344,Z 167,A -54.3826,B 10.3441,C 0.3427,E1 10.4391,E2 505.5495} C_DIS
LIN {X 75.231,Y -118.8107,Z 167,A -56.1387,B 10.344,C 0.3437,E1 10.435,E2 507.2965} C_DIS
LIN {X 71.5547,Y -121.0608,Z 167,A -57.8861,B 10.3439,C 0.3464,E1 10.4308,E2 509.0444} C_DIS
LIN {X 67.8082,Y -123.1984,Z 167,A -59.5914,B 10.3439,C 0.3478,E1 10.4267,E2 510.7444} C_DIS
LIN {X 64.5476,Y -124.9376,Z 167,A -61.1977,B 10.3437,C 0.3525,E1 10.4227,E2 512.3652} C_DIS
LIN {X 60.9106,Y -126.7482,Z 167,A -62.7233,B 10.3437,C 0.3516,E1 10.4189,E2 513.8753} C_DIS
LIN {X 57.7701,Y -128.2103,Z 167,A -64.1492,B 10.3437,C 0.3538,E1 10.4153,E2 515.3043} C_DIS
LIN {X 54.4963,Y -129.6355,Z 167,A -65.5774,B 10.3436,C 0.355,E1 10.4116,E2 516.7302} C_DIS
LIN {X 51.264,Y -130.9475,Z 167,A -66.9897,B 10.3436,C 0.3565,E1 10.4079,E2 518.1425} C_DIS
LIN {X 47.8782,Y -132.2227,Z 167,A -68.4203,B 10.3436,C 0.3571,E1 10.4042,E2 519.5686} C_DIS
LIN {X 44.4845,Y -133.4027,Z 167,A -69.9703,B 10.3434,C 0.3608,E1 10.4001,E2 521.1309} C_DIS
LIN {X 40.4467,Y -134.6829,Z 167,A -71.5921,B 10.3434,C 0.3599,E1 10.3958,E2 522.7405} C_DIS
LIN {X 36.6374,Y -135.7678,Z 167,A -73.2536,B 10.3434,C 0.3625,E1 10.3913,E2 524.4093} C_DIS
LIN {X 33.1915,Y -136.6512,Z 167,A -74.6745,B 10.3434,C 0.3631,E1 10.3874,E2 525.8276} C_DIS
LIN {X 29.872,Y -137.415,Z 167,A -76.0551,B 10.3433,C 0.364,E1 10.3837,E2 527.2082} C_DIS
LIN {X 26.5545,Y -138.0944,Z 167,A -77.4273,B 10.3433,C 0.3647,E1 10.3799,E2 528.5803} C_DIS
LIN {X 23.2546,Y -138.6882,Z 167,A -78.6989,B 10.3433,C 0.3633,E1 10.3765,E2 529.8405} C_DIS
LIN {X 20.2456,Y -139.1598,Z 167,A -80.0398,B 10.3433,C 0.3664,E1 10.3727,E2 531.1952} C_DIS
LIN {X 17.2175,Y -139.5675,Z 167,A -81.2864,B 10.3432,C 0.3671,E1 10.3693,E2 532.4428} C_DIS
LIN {X 13.7917,Y -139.9469,Z 167,A -82.6842,B 10.3432,C 0.3675,E1 10.3654,E2 533.8406} C_DIS
LIN {X 9.7877,Y -140.2836,Z 167,A -84.4314,B 10.343,C 0.3707,E1 10.3605,E2 535.603} C_DIS
LIN {X 5.178,Y -140.5295,Z 167,A -86.1935,B 10.3431,C 0.3684,E1 10.3556,E2 537.3507} C_DIS
LIN {X 1.6213,Y -140.617,Z 167,A -87.7365,B 10.3431,C 0.3709,E1 10.3513,E2 538.9066} C_DIS
LIN {X 1.6213,Y -140.617,Z 167,A -87.7365,B 10.3431,C 0.3709,E1 10.3513,E2 538.9066} C_DIS
Enddeposition()
LIN {X 0.9547,Y -131.6551,Z 168,A -87.8641,B 10.6484,C 0.2926,E1 10.655,E2 538.5781} C_DIS
Startdeposition()
$VEL.CP = VEL_PRINT
LIN {X 4.1942,Y -131.596,Z 168,A -86.1141,B 10.6486,C 0.2847,E1 10.66,E2 536.7861} C_DIS
LIN {X 8.0736,Y -131.4139,Z 168,A -84.5773,B 10.6486,C 0.2877,E1 10.6642,E2 535.267} C_DIS
LIN {X 11.2927,Y -131.1766,Z 168,A -83.1809,B 10.6486,C 0.2873,E1 10.6681,E2 533.8709} C_DIS
LIN {X 15.13,Y -130.7901,Z 168,A -81.4905,B 10.6486,C 0.2863,E1 10.6728,E2 532.1781} C_DIS
LIN {X 19.3203,Y -130.2381,Z 168,A -79.6742,B 10.6486,C 0.2859,E1 10.6778,E2 530.3635} C_DIS
LIN {X 22.5073,Y -129.7253,Z 168,A -78.0996,B 10.6487,C 0.2811,E1 10.6822,E2 528.7673} C_DIS
LIN {X 26.6405,Y -128.9386,Z 168,A -76.323,B 10.6487,C 0.2811,E1 10.6871,E2 526.996} C_DIS
LIN {X 30.7033,Y -128.0314,Z 168,A -74.7197,B 10.6487,C 0.2845,E1 10.6914,E2 525.4168} C_DIS
LIN {X 34.0137,Y -127.1919,Z 168,A -73.0868,B 10.6487,C 0.2798,E1 10.6958,E2 523.7649} C_DIS
LIN {X 38.2187,Y -125.9926,Z 168,A -71.2602,B 10.6487,C 0.2798,E1 10.7007,E2 521.9463} C_DIS
LIN {X 41.2894,Y -125.0199,Z 168,A -69.8664,B 10.6488,C 0.2785,E1 10.7044,E2 520.5524} C_DIS
LIN {X 44.3557,Y -123.9651,Z 168,A -68.4625,B 10.6488,C 0.2771,E1 10.7081,E2 519.1482} C_DIS
LIN {X 47.38,Y -122.8411,Z 168,A -67.067,B 10.6488,C 0.2757,E1 10.7118,E2 517.7527} C_DIS
LIN {X 50.3755,Y -121.6435,Z 168,A -65.6725,B 10.6489,C 0.2742,E1 10.7154,E2 516.3582} C_DIS
LIN {X 53.4493,Y -120.3243,Z 168,A -64.2628,B 10.6489,C 0.2734,E1 10.719,E2 514.9529} C_DIS
LIN {X 56.2918,Y -119.0216,Z 168,A -62.8536,B 10.649,C 0.2705,E1 10.7226,E2 513.5365} C_DIS
LIN {X 59.2041,Y -117.6005,Z 168,A -61.477,B 10.649,C 0.2693,E1 10.726,E2 512.1628} C_DIS
LIN {X 62.0717,Y -116.1136,Z 168,A -59.954,B 10.6492,C 0.2644,E1 10.7298,E2 510.6242} C_DIS
LIN {X 65.4497,Y -114.2435,Z 168,A -58.3446,B 10.6492,C 0.2635,E1 10.7337,E2 509.022} C_DIS
LIN {X 69.0661,Y -112.0942,Z 168,A -56.587,B 10.6492,C 0.2623,E1 10.7379,E2 507.2716} C_DIS
LIN {X 72.3398,Y -110.0097,Z 168,A -54.9175,B 10.6492,C 0.2599,E1 10.7418,E2 505.6029} C_DIS
LIN {X 75.2955,Y -108.0082,Z 168,A -53.2548,B 10.6494,C 0.2545,E1 10.7456,E2 503.9253} C_DIS
LIN {X 78.4272,Y -105.7564,Z 168,A -51.6132,B 10.6494,C 0.2523,E1 10.7493,E2 502.2865} C_DIS
LIN {X 81.6274,Y -103.3068,Z 168,A -49.8663,B 10.6495,C 0.2492,E1 10.7532,E2 500.5388} C_DIS
LIN {X 85.0151,Y -100.5372,Z 168,A -47.9824,B 10.6495,C 0.2459,E1 10.7572,E2 498.6555} C_DIS
LIN {X 88.1791,Y -97.7741,Z 168,A -46.2029,B 10.6497,C 0.2434,E1 10.7609,E2 496.88} C_DIS
LIN {X 91.0031,Y -95.1505,Z 168,A -44.5374,B 10.6497,C 0.2401,E1 10.7643,E2 495.2141} C_DIS
LIN {X 93.9905,Y -92.2006,Z 168,A -42.7456,B 10.6497,C 0.2371,E1 10.7679,E2 493.4247} C_DIS
LIN {X 96.7941,Y -89.2531,Z 168,A -40.9911,B 10.6499,C 0.2335,E1 10.7712,E2 491.6703} C_DIS
LIN {X 99.4809,Y -86.249,Z 168,A -39.1863,B 10.6499,C 0.2283,E1 10.7745,E2 489.8574} C_DIS
LIN {X 102.2713,Y -82.9209,Z 168,A -37.3425,B 10.6501,C 0.225,E1 10.7778,E2 488.0172} C_DIS
LIN {X 104.7813,Y -79.7255,Z 168,A -35.5735,B 10.6501,C 0.2208,E1 10.7808,E2 486.2462} C_DIS
LIN {X 107.0713,Y -76.6219,Z 168,A -34.0467,B 10.6501,C 0.2205,E1 10.7833,E2 484.7359} C_DIS
LIN {X 109.1098,Y -73.6902,Z 168,A -32.503,B 10.6502,C 0.2169,E1 10.7857,E2 483.1918} C_DIS
LIN {X 111.2365,Y -70.439,Z 168,A -30.7262,B 10.6503,C 0.2104,E1 10.7884,E2 481.4026} C_DIS
LIN {X 113.2546,Y -67.1466,Z 168,A -29.1096,B 10.6504,C 0.2077,E1 10.7908,E2 479.792} C_DIS
LIN {X 115.3756,Y -63.4335,Z 168,A -27.3294,B 10.6504,C 0.2049,E1 10.7932,E2 478.0195} C_DIS
LIN {X 117.1442,Y -60.1003,Z 168,A -25.7333,B 10.6505,C 0.2017,E1 10.7953,E2 476.427} C_DIS
LIN {X 118.5538,Y -57.2711,Z 168,A -24.3902,B 10.6505,C 0.1988,E1 10.7969,E2 475.0864} C_DIS
LIN {X 119.9682,Y -54.2456,Z 168,A -22.9316,B 10.6506,C 0.1947,E1 10.7986,E2 473.6255} C_DIS
LIN {X 121.3953,Y -50.9696,Z 168,A -21.5082,B 10.6506,C 0.1938,E1 10.8002,E2 472.2163} C_DIS
LIN {X 122.4821,Y -48.3033,Z 168,A -20.0418,B 10.6508,C 0.185,E1 10.8017,E2 470.7226} C_DIS
LIN {X 123.9651,Y -44.3557,Z 168,A -18.3447,B 10.6508,C 0.1833,E1 10.8033,E2 469.0402} C_DIS
LIN {X 125.22,Y -40.6823,Z 168,A -16.5816,B 10.651,C 0.1767,E1 10.8049,E2 467.2663} C_DIS
LIN {X 126.273,Y -37.2818,Z 168,A -15.0322,B 10.651,C 0.1723,E1 10.8061,E2 465.7152} C_DIS
LIN {X 127.5004,Y -32.8416,Z 168,A -13.1153,B 10.651,C 0.1688,E1 10.8075,E2 463.8067} C_DIS
LIN {X 128.2332,Y -29.8541,Z 168,A -11.8488,B 10.6511,C 0.1668,E1 10.8083,E2 462.5475} C_DIS
LIN {X 128.9372,Y -26.6475,Z 168,A -10.3611,B 10.6511,C 0.1612,E1 10.8092,E2 461.051} C_DIS
LIN {X 129.7265,Y -22.5004,Z 168,A -8.643,B 10.6512,C 0.1589,E1 10.8101,E2 459.3454} C_DIS
LIN {X 130.239,Y -19.314,Z 168,A -7.2337,B 10.6512,C 0.1546,E1 10.8107,E2 457.934} C_DIS
LIN {X 130.6726,Y -16.1158,Z 168,A -5.7203,B 10.6514,C 0.1478,E1 10.8112,E2 456.406} C_DIS
LIN {X 131.0882,Y -12.2776,Z 168,A -4.2138,B 10.6514,C 0.1472,E1 10.8116,E2 454.9187} C_DIS
LIN {X 131.3743,Y -8.715,Z 168,A -2.6997,B 10.6514,C 0.1437,E1 10.8119,E2 453.408} C_DIS
LIN {X 131.5729,Y -4.8421,Z 168,A -1.019,B 10.6515,C 0.139,E1 10.8121,E2 451.7263} C_DIS
LIN {X 131.653,Y -1.6163,Z 168,A 0.3881,B 10.6515,C 0.1348,E1 10.8122,E2 450.3175} C_DIS
LIN {X 131.6426,Y 2.2448,Z 168,A 2.0739,B 10.6516,C 0.1297,E1 10.8122,E2 448.6293} C_DIS
LIN {X 131.5029,Y 6.4652,Z 168,A 3.8505,B 10.6516,C 0.1259,E1 10.812,E2 446.8582} C_DIS
LIN {X 131.3048,Y 9.6874,Z 168,A 5.2287,B 10.6517,C 0.1224,E1 10.8117,E2 445.4818} C_DIS
LIN {X 131.0281,Y 12.9038,Z 168,A 6.7306,B 10.6517,C 0.1159,E1 10.8113,E2 443.9669} C_DIS
LIN {X 130.5937,Y 16.7387,Z 168,A 8.2855,B 10.6517,C 0.1142,E1 10.8108,E2 442.4254} C_DIS
LIN {X 129.9908,Y 20.9216,Z 168,A 10.0994,B 10.6518,C 0.1095,E1 10.81,E2 440.6129} C_DIS
LIN {X 129.3191,Y 24.7243,Z 168,A 11.7966,B 10.6519,C 0.1042,E1 10.8092,E2 438.912} C_DIS
LIN {X 128.464,Y 28.8437,Z 168,A 13.6814,B 10.6519,C 0.0977,E1 10.8081,E2 437.0192} C_DIS
LIN {X 127.5589,Y 32.6111,Z 168,A 15.3241,B 10.6519,C 0.094,E1 10.8069,E2 435.3802} C_DIS
LIN {X 126.2752,Y 37.274,Z 168,A 17.2897,B 10.652,C 0.0916,E1 10.8055,E2 433.4296} C_DIS
LIN {X 125.2324,Y 40.6435,Z 168,A 18.9627,B 10.652,C 0.0839,E1 10.804,E2 431.7387} C_DIS
LIN {X 123.9659,Y 44.3535,Z 168,A 20.4896,B 10.652,C 0.0837,E1 10.8026,E2 430.2319} C_DIS
LIN {X 122.8422,Y 47.377,Z 168,A 21.8743,B 10.6521,C 0.0804,E1 10.8013,E2 428.8485} C_DIS
LIN {X 121.6453,Y 50.3712,Z 168,A 23.2983,B 10.6521,C 0.0761,E1 10.7998,E2 427.4209} C_DIS
LIN {X 120.3662,Y 53.3557,Z 168,A 24.6531,B 10.6521,C 0.0738,E1 10.7983,E2 426.072} C_DIS
LIN {X 119.0218,Y 56.2914,Z 168,A 26.0394,B 10.6521,C 0.0705,E1 10.7966,E2 424.687} C_DIS
LIN {X 117.5994,Y 59.2062,Z 168,A 27.4297,B 10.6521,C 0.0674,E1 10.7949,E2 423.2982} C_DIS
LIN {X 116.1172,Y 62.0649,Z 168,A 28.9418,B 10.6522,C 0.0611,E1 10.7929,E2 421.7719} C_DIS
LIN {X 114.2556,Y 65.4285,Z 168,A 30.5327,B 10.6522,C 0.0589,E1 10.7907,E2 420.1898} C_DIS
LIN {X 112.112,Y 69.0371,Z 168,A 32.2895,B 10.6522,C 0.0561,E1 10.7882,E2 418.4402} C_DIS
LIN {X 110.0155,Y 72.331,Z 168,A 33.9575,B 10.6522,C 0.0527,E1 10.7857,E2 416.7749} C_DIS
LIN {X 108.0116,Y 75.2906,Z 168,A 35.6204,B 10.6523,C 0.0464,E1 10.783,E2 415.0983} C_DIS
LIN {X 105.6817,Y 78.5275,Z 168,A 37.3339,B 10.6523,C 0.0429,E1 10.7802,E2 413.3864} C_DIS
LIN {X 102.8348,Y 82.2209,Z 168,A 39.3286,B 10.6523,C 0.0391,E1 10.7768,E2 411.3949} C_DIS
LIN {X 100.1812,Y 85.4339,Z 168,A 41.0544,B 10.6523,C 0.0373,E1 10.7737,E2 409.6786} C_DIS
LIN {X 97.5508,Y 88.4252,Z 168,A 42.8153,B 10.6523,C 0.0329,E1 10.7704,E2 407.9137} C_DIS
LIN {X 94.5748,Y 91.6012,Z 168,A 44.6839,B 10.6523,C 0.0295,E1 10.7668,E2 406.0474} C_DIS
LIN {X 91.5999,Y 94.5761,Z 168,A 46.5318,B 10.6523,C 0.0254,E1 10.7631,E2 404.1967} C_DIS
LIN {X 88.4244,Y 97.5515,Z 168,A 48.3764,B 10.6523,C 0.0229,E1 10.7594,E2 402.3573} C_DIS
LIN {X 85.0685,Y 100.4918,Z 168,A 50.296,B 10.6523,C 0.0198,E1 10.7553,E2 400.4398} C_DIS
LIN {X 81.8768,Y 103.1086,Z 168,A 52.0484,B 10.6523,C 0.0176,E1 10.7515,E2 398.692} C_DIS
LIN {X 79.2152,Y 105.1672,Z 168,A 53.4531,B 10.6523,C 0.0165,E1 10.7484,E2 397.2941} C_DIS
LIN {X 76.6203,Y 107.0725,Z 168,A 54.8394,B 10.6523,C 0.0145,E1 10.7453,E2 395.9092} C_DIS
LIN {X 73.6939,Y 109.1073,Z 168,A 56.503,B 10.6524,C 0.0094,E1 10.7414,E2 394.2319} C_DIS
LIN {X 69.9037,Y 111.5743,Z 168,A 58.3376,B 10.6524,C 0.0094,E1 10.7371,E2 392.4129} C_DIS
LIN {X 67.1472,Y 113.2542,Z 168,A 59.804,B 10.6524,C 0.006,E1 10.7336,E2 390.939} C_DIS
LIN {X 63.4834,Y 115.348,Z 168,A 61.6944,B 10.6524,C 0.0022,E1 10.729,E2 389.0421} C_DIS
LIN {X 60.0781,Y 117.1555,Z 168,A 63.215,B 10.6524,C 0.0036,E1 10.7252,E2 387.5399} C_DIS
LIN {X 56.8373,Y 118.761,Z 168,A 64.6735,B 10.6524,C 0.0043,E1 10.7216,E2 386.0949} C_DIS
LIN {X 54.2523,Y 119.9652,Z 168,A 66.099,B 10.6524,C -0.0014,E1 10.7179,E2 384.6477} C_DIS
LIN {X 50.3873,Y 121.6385,Z 168,A 67.9454,B 10.6524,C -0.0037,E1 10.7132,E2 382.7997} C_DIS
LIN {X 46.7886,Y 123.0688,Z 168,A 69.618,B 10.6524,C -0.0051,E1 10.7088,E2 381.1288} C_DIS
LIN {X 43.7606,Y 124.1778,Z 168,A 71.017,B 10.6524,C -0.0064,E1 10.7052,E2 379.7304} C_DIS
LIN {X 40.7066,Y 125.2123,Z 168,A 72.4377,B 10.6524,C -0.008,E1 10.7014,E2 378.3079} C_DIS
LIN {X 36.6762,Y 126.4502,Z 168,A 74.1396,B 10.6524,C -0.0064,E1 10.6969,E2 376.6219} C_DIS
LIN {X 32.8847,Y 127.4895,Z 168,A 75.926,B 10.6524,C -0.0093,E1 10.692,E2 374.8269} C_DIS
LIN {X 29.8017,Y 128.2452,Z 168,A 77.2288,B 10.6524,C -0.0084,E1 10.6885,E2 373.5337} C_DIS
LIN {X 26.6486,Y 128.937,Z 168,A 78.708,B 10.6524,C -0.0109,E1 10.6845,E2 372.0461} C_DIS
LIN {X 22.5123,Y 129.7244,Z 168,A 80.4412,B 10.6524,C -0.0096,E1 10.6797,E2 370.3251} C_DIS
LIN {X 19.3242,Y 130.2376,Z 168,A 81.8715,B 10.6524,C -0.0107,E1 10.6758,E2 368.8923} C_DIS
LIN {X 16.1158,Y 130.6726,Z 168,A 83.405,B 10.6524,C -0.0139,E1 10.6715,E2 367.3445} C_DIS
LIN {X 12.2752,Y 131.0885,Z 168,A 84.9315,B 10.6524,C -0.0109,E1 10.6673,E2 365.8368} C_DIS
LIN {X 8.7138,Y 131.3744,Z 168,A 86.4217,B 10.6524,C -0.0098,E1 10.6632,E2 364.3547} C_DIS
LIN {X 5.4909,Y 131.5476,Z 168,A 87.8073,B 10.6524,C -0.0095,E1 10.6593,E2 362.9719} C_DIS
LIN {X 2.2491,Y 131.6425,Z 168,A 89.3875,B 10.6524,C -0.0132,E1 10.6548,E2 361.3726} C_DIS
LIN {X -2.2439,Y 131.6425,Z 168,A 91.3126,B 10.6524,C -0.0124,E1 10.6495,E2 359.4519} C_DIS
LIN {X -6.4517,Y 131.5036,Z 168,A 93.1031,B 10.6524,C -0.0112,E1 10.6445,E2 357.6672} C_DIS
LIN {X -9.6867,Y 131.3048,Z 168,A 94.5077,B 10.6524,C -0.0108,E1 10.6406,E2 356.264} C_DIS
LIN {X -12.9032,Y 131.0282,Z 168,A 96.0334,B 10.6524,C -0.0129,E1 10.6363,E2 354.725} C_DIS
LIN {X -16.7403,Y 130.5935,Z 168,A 97.6091,B 10.6524,C -0.01,E1 10.632,E2 353.1625} C_DIS
LIN {X -19.3732,Y 130.2306,Z 168,A 98.7525,B 10.6524,C -0.0092,E1 10.6288,E2 352.0215} C_DIS
LIN {X -22.51,Y 129.7248,Z 168,A 100.3145,B 10.6524,C -0.0123,E1 10.6245,E2 350.4393} C_DIS
LIN {X -26.6459,Y 128.9375,Z 168,A 102.1094,B 10.6524,C -0.0103,E1 10.6196,E2 348.6499} C_DIS
LIN {X -30.4325,Y 128.0967,Z 168,A 103.8146,B 10.6524,C -0.0095,E1 10.6149,E2 346.9438} C_DIS
LIN {X -34.1673,Y 127.151,Z 168,A 105.3607,B 10.6524,C -0.0055,E1 10.6108,E2 345.4141} C_DIS
LIN {X -37.2841,Y 126.2723,Z 168,A 106.7738,B 10.6524,C -0.0044,E1 10.607,E2 344.0016} C_DIS
LIN {X -40.6611,Y 125.2268,Z 168,A 108.4795,B 10.6524,C -0.0064,E1 10.6024,E2 342.2774} C_DIS
LIN {X -44.3493,Y 123.9674,Z 168,A 110.0292,B 10.6524,C -0.0016,E1 10.5984,E2 340.7462} C_DIS
LIN {X -47.3849,Y 122.8392,Z 168,A 111.4423,B 10.6524,C -0.0002,E1 10.5947,E2 339.3337} C_DIS
LIN {X -50.3811,Y 121.6411,Z 168,A 112.8537,B 10.6524,C 0.0013,E1 10.591,E2 337.9227} C_DIS
LIN {X -53.3478,Y 120.3697,Z 168,A 114.2743,B 10.6524,C 0.0026,E1 10.5874,E2 336.5013} C_DIS
LIN {X -56.3031,Y 119.0162,Z 168,A 115.8144,B 10.6524,C 0.0019,E1 10.5835,E2 334.9477} C_DIS
LIN {X -59.3068,Y 117.5482,Z 168,A 117.1024,B 10.6524,C 0.0072,E1 10.5803,E2 333.6805} C_DIS
LIN {X -62.1895,Y 116.0503,Z 168,A 118.6625,B 10.6524,C 0.0063,E1 10.5764,E2 332.1046} C_DIS
LIN {X -65.3785,Y 114.2841,Z 168,A 120.2252,B 10.6524,C 0.0091,E1 10.5726,E2 330.5461} C_DIS
LIN {X -69.0676,Y 112.0933,Z 168,A 122.0633,B 10.6524,C 0.0126,E1 10.5682,E2 328.7131} C_DIS
LIN {X -72.34,Y 110.0096,Z 168,A 123.7587,B 10.6524,C 0.0152,E1 10.5643,E2 327.0184} C_DIS
LIN {X -75.2969,Y 108.0072,Z 168,A 125.4516,B 10.6524,C 0.0151,E1 10.5603,E2 325.3107} C_DIS
LIN {X -78.4321,Y 105.7527,Z 168,A 127.1228,B 10.6524,C 0.0182,E1 10.5566,E2 323.6422} C_DIS
LIN {X -81.634,Y 103.3016,Z 168,A 128.9041,B 10.6524,C 0.021,E1 10.5527,E2 321.8596} C_DIS
LIN {X -85.0151,Y 100.5371,Z 168,A 130.8192,B 10.6524,C 0.0243,E1 10.5485,E2 319.9446} C_DIS
LIN {X -88.1836,Y 97.7701,Z 168,A 132.6358,B 10.6524,C 0.0282,E1 10.5448,E2 318.1316} C_DIS
LIN {X -91.0114,Y 95.1425,Z 168,A 134.3395,B 10.6524,C 0.0312,E1 10.5413,E2 316.4268} C_DIS
LIN {X -94.0169,Y 92.1738,Z 168,A 136.1706,B 10.6524,C 0.0352,E1 10.5377,E2 314.5984} C_DIS
LIN {X -96.7966,Y 89.2504,Z 168,A 137.9554,B 10.6524,C 0.0385,E1 10.5343,E2 312.812} C_DIS
LIN {X -99.4858,Y 86.2434,Z 168,A 139.8026,B 10.6524,C 0.0406,E1 10.5309,E2 310.9559} C_DIS
LIN {X -102.29,Y 82.8976,Z 168,A 141.6896,B 10.6524,C 0.0452,E1 10.5275,E2 309.0725} C_DIS
LIN {X -104.7824,Y 79.7241,Z 168,A 143.4958,B 10.6523,C 0.0484,E1 10.5244,E2 307.2623} C_DIS
LIN {X -107.0744,Y 76.6176,Z 168,A 145.0592,B 10.6523,C 0.0547,E1 10.5219,E2 305.7144} C_DIS
LIN {X -109.1146,Y 73.6831,Z 168,A 146.6457,B 10.6523,C 0.0579,E1 10.5194,E2 304.1259} C_DIS
LIN {X -111.2482,Y 70.4205,Z 168,A 148.4665,B 10.6523,C 0.0597,E1 10.5166,E2 302.2924} C_DIS
LIN {X -113.2655,Y 67.1284,Z 168,A 150.1266,B 10.6523,C 0.0644,E1 10.5142,E2 300.6365} C_DIS
LIN {X -115.3487,Y 63.4821,Z 168,A 151.908,B 10.6522,C 0.07,E1 10.5118,E2 298.8625} C_DIS
LIN {X -117.1571,Y 60.075,Z 168,A 153.5986,B 10.6522,C 0.0742,E1 10.5096,E2 297.1723} C_DIS
LIN {X -118.5931,Y 57.1889,Z 168,A 155.0256,B 10.6522,C 0.0774,E1 10.5079,E2 295.7441} C_DIS
LIN {X -119.9614,Y 54.2606,Z 168,A 156.4705,B 10.6522,C 0.0805,E1 10.5062,E2 294.2962} C_DIS
LIN {X -121.3796,Y 51.0072,Z 168,A 157.9101,B 10.6521,C 0.0867,E1 10.5046,E2 292.8707} C_DIS
LIN {X -122.5856,Y 48.0371,Z 168,A 159.4866,B 10.6521,C 0.0871,E1 10.503,E2 291.2743} C_DIS
LIN {X -123.9679,Y 44.3479,Z 168,A 161.1674,B 10.6521,C 0.0925,E1 10.5013,E2 289.5994} C_DIS
LIN {X -125.2168,Y 40.6924,Z 168,A 162.9736,B 10.652,C 0.0948,E1 10.4997,E2 287.7803} C_DIS
LIN {X -126.2734,Y 37.2801,Z 168,A 164.5695,B 10.652,C 0.0984,E1 10.4985,E2 286.1813} C_DIS
LIN {X -127.3125,Y 33.5615,Z 168,A 166.1482,B 10.6519,C 0.1051,E1 10.4973,E2 284.6163} C_DIS
LIN {X -128.2409,Y 29.8202,Z 168,A 167.8683,B 10.6519,C 0.1091,E1 10.4962,E2 282.8931} C_DIS
LIN {X -128.9383,Y 26.6423,Z 168,A 169.3704,B 10.6519,C 0.1116,E1 10.4953,E2 281.3823} C_DIS
LIN {X -129.721,Y 22.531,Z 168,A 171.1866,B 10.6518,C 0.117,E1 10.4944,E2 279.5687} C_DIS
LIN {X -130.231,Y 19.37,Z 168,A 172.5579,B 10.6518,C 0.1214,E1 10.4938,E2 278.2015} C_DIS
LIN {X -130.663,Y 16.1959,Z 168,A 174.1051,B 10.6518,C 0.1226,E1 10.4933,E2 276.6377} C_DIS
LIN {X -131.0896,Y 12.2638,Z 168,A 175.699,B 10.6516,C 0.13,E1 10.4928,E2 275.0606} C_DIS
LIN {X -131.3754,Y 8.6981,Z 168,A 177.2076,B 10.6516,C 0.1355,E1 10.4925,E2 273.5594} C_DIS
LIN {X -131.5728,Y 4.8447,Z 168,A 178.9787,B 10.6516,C 0.1387,E1 10.4923,E2 271.7791} C_DIS
LIN {X -131.6531,Y 1.6148,Z 168,A -179.5716,B 10.6515,C 0.142,E1 10.4923,E2 270.3257} C_DIS
LIN {X -131.6424,Y -2.2576,Z 168,A -177.8349,B 10.6515,C 0.1459,E1 10.4923,E2 268.5846} C_DIS
LIN {X -131.5029,Y -6.4645,Z 168,A -176.0116,B 10.6513,C 0.1515,E1 10.4925,E2 266.7641} C_DIS
LIN {X -131.3048,Y -9.6876,Z 168,A -174.5934,B 10.6513,C 0.1553,E1 10.4927,E2 265.3457} C_DIS
LIN {X -131.028,Y -12.905,Z 168,A -173.0442,B 10.6513,C 0.1567,E1 10.4931,E2 263.7808} C_DIS
LIN {X -130.5917,Y -16.7537,Z 168,A -171.4477,B 10.6512,C 0.1632,E1 10.4937,E2 262.1964} C_DIS
LIN {X -129.9509,Y -21.1609,Z 168,A -169.3789,B 10.6512,C 0.1664,E1 10.4945,E2 260.114} C_DIS
LIN {X -129.3148,Y -24.7468,Z 168,A -167.8322,B 10.651,C 0.1716,E1 10.4953,E2 258.5732} C_DIS
LIN {X -128.4635,Y -28.8458,Z 168,A -166.0314,B 10.651,C 0.1772,E1 10.4964,E2 256.7765} C_DIS
LIN {X -127.5669,Y -32.5796,Z 168,A -164.3425,B 10.6509,C 0.1816,E1 10.4975,E2 255.087} C_DIS
LIN {X -126.7221,Y -35.7252,Z 168,A -162.9044,B 10.6509,C 0.1851,E1 10.4986,E2 253.6475} C_DIS
LIN {X -125.8024,Y -38.8403,Z 168,A -161.4382,B 10.6508,C 0.1881,E1 10.4998,E2 252.1763} C_DIS
LIN {X -124.5003,Y -42.8307,Z 168,A -159.6195,B 10.6507,C 0.1932,E1 10.5014,E2 250.3601} C_DIS
LIN {X -123.4128,Y -45.8702,Z 168,A -158.197,B 10.6507,C 0.1967,E1 10.5027,E2 248.9365} C_DIS
LIN {X -122.13,Y -49.1826,Z 168,A -156.5723,B 10.6506,C 0.1993,E1 10.5044,E2 247.3035} C_DIS
LIN {X -120.6121,Y -52.799,Z 168,A -154.7702,B 10.6506,C 0.202,E1 10.5064,E2 245.4914} C_DIS
LIN {X -119.033,Y -56.268,Z 168,A -153.2344,B 10.6504,C 0.2087,E1 10.5082,E2 243.9715} C_DIS
LIN {X -117.6036,Y -59.198,Z 168,A -151.7914,B 10.6504,C 0.2119,E1 10.51,E2 242.5265} C_DIS
LIN {X -116.1189,Y -62.0617,Z 168,A -150.2386,B 10.6504,C 0.2126,E1 10.512,E2 240.957} C_DIS
LIN {X -114.2525,Y -65.4339,Z 168,A -148.6031,B 10.6502,C 0.2176,E1 10.5143,E2 239.3275} C_DIS
LIN {X -112.0911,Y -69.0712,Z 168,A -146.7975,B 10.6502,C 0.2228,E1 10.5169,E2 237.5273} C_DIS
LIN {X -110.0084,Y -72.3417,Z 168,A -145.0966,B 10.65,C 0.2266,E1 10.5195,E2 235.8258} C_DIS
LIN {X -108.0071,Y -75.2971,Z 168,A -143.5218,B 10.65,C 0.2298,E1 10.522,E2 234.2493} C_DIS
LIN {X -105.7556,Y -78.4283,Z 168,A -141.7259,B 10.65,C 0.2314,E1 10.5249,E2 232.4402} C_DIS
LIN {X -103.3059,Y -81.6285,Z 168,A -139.9435,B 10.6498,C 0.2347,E1 10.528,E2 230.6553} C_DIS
LIN {X -100.5341,Y -85.0187,Z 168,A -138.0201,B 10.6498,C 0.2385,E1 10.5314,E2 228.7306} C_DIS
LIN {X -97.7658,Y -88.1883,Z 168,A -136.2015,B 10.6497,C 0.2427,E1 10.5348,E2 226.9144} C_DIS
LIN {X -95.1373,Y -91.0169,Z 168,A -134.496,B 10.6497,C 0.2456,E1 10.5381,E2 225.2066} C_DIS
LIN {X -92.1795,Y -94.0112,Z 168,A -132.6733,B 10.6495,C 0.2494,E1 10.5417,E2 223.3856} C_DIS
LIN {X -89.2556,Y -96.7918,Z 168,A -130.8613,B 10.6495,C 0.2517,E1 10.5454,E2 221.5675} C_DIS
LIN {X -86.226,Y -99.5008,Z 168,A -129.037,B 10.6495,C 0.2538,E1 10.5492,E2 219.737} C_DIS
LIN {X -82.896,Y -102.2913,Z 168,A -127.1619,B 10.6493,C 0.2575,E1 10.5533,E2 217.8643} C_DIS
LIN {X -79.726,Y -104.7809,Z 168,A -125.3644,B 10.6493,C 0.2595,E1 10.5572,E2 216.062} C_DIS
LIN {X -76.6249,Y -107.0691,Z 168,A -123.809,B 10.6492,C 0.2648,E1 10.5607,E2 214.5216} C_DIS
LIN {X -73.6961,Y -109.1058,Z 168,A -122.2357,B 10.6492,C 0.2668,E1 10.5644,E2 212.9461} C_DIS
LIN {X -70.4413,Y -111.2351,Z 168,A -120.3964,B 10.6492,C 0.2662,E1 10.5687,E2 211.0894} C_DIS
LIN {X -67.1381,Y -113.2596,Z 168,A -118.7683,B 10.649,C 0.2698,E1 10.5726,E2 209.4684} C_DIS
LIN {X -63.4894,Y -115.3446,Z 168,A -116.9953,B 10.649,C 0.2734,E1 10.5769,E2 207.7023} C_DIS
LIN {X -60.0836,Y -117.1527,Z 168,A -115.3107,B 10.6489,C 0.2753,E1 10.5811,E2 206.017} C_DIS
LIN {X -57.1791,Y -118.5977,Z 168,A -113.7718,B 10.6489,C 0.2743,E1 10.585,E2 204.4627} C_DIS
LIN {X -53.358,Y -120.3651,Z 168,A -111.8981,B 10.6489,C 0.2754,E1 10.5897,E2 202.5839} C_DIS
LIN {X -49.7928,Y -121.8841,Z 168,A -110.3652,B 10.6488,C 0.2804,E1 10.5937,E2 201.0696} C_DIS
LIN {X -46.7927,Y -123.0672,Z 168,A -108.8453,B 10.6488,C 0.2792,E1 10.5977,E2 199.5355} C_DIS
LIN {X -43.7666,Y -124.1758,Z 168,A -107.3968,B 10.6488,C 0.2795,E1 10.6015,E2 198.0813} C_DIS
LIN {X -40.7024,Y -125.2136,Z 168,A -106.0221,B 10.6488,C 0.2813,E1 10.6051,E2 196.7104} C_DIS
LIN {X -36.4499,Y -126.5165,Z 168,A -104.1973,B 10.6486,C 0.2851,E1 10.61,E2 194.8987} C_DIS
LIN {X -33.5524,Y -127.3149,Z 168,A -102.8717,B 10.6486,C 0.2855,E1 10.6135,E2 193.5706} C_DIS
LIN {X -29.8046,Y -128.2445,Z 168,A -101.1783,B 10.6486,C 0.2862,E1 10.6181,E2 191.8753} C_DIS
LIN {X -26.6498,Y -128.9367,Z 168,A -99.6747,B 10.6486,C 0.2847,E1 10.6223,E2 190.3594} C_DIS
LIN {X -22.5163,Y -129.7237,Z 168,A -97.9516,B 10.6486,C 0.2878,E1 10.627,E2 188.649} C_DIS
LIN {X -19.3173,Y -130.2386,Z 168,A -96.515,B 10.6486,C 0.2877,E1 10.631,E2 187.2087} C_DIS
LIN {X -16.1172,Y -130.6724,Z 168,A -94.9779,B 10.6486,C 0.2851,E1 10.6353,E2 185.6551} C_DIS
LIN {X -12.2797,Y -131.088,Z 168,A -93.4493,B 10.6486,C 0.2887,E1 10.6395,E2 184.1442} C_DIS
LIN {X -8.7198,Y -131.374,Z 168,A -91.8764,B 10.6486,C 0.2885,E1 10.6439,E2 182.5685} C_DIS
LIN {X -4.8459,Y -131.5728,Z 168,A -90.209,B 10.6486,C 0.2889,E1 10.6485,E2 180.9028} C_DIS
LIN {X -1.6202,Y -131.653,Z 168,A -88.7692,B 10.6486,C 0.288,E1 10.6525,E2 179.4581} C_DIS
LIN {X 0.9547,Y -131.6551,Z 168,A -87.8637,B 10.6484,C 0.2927,E1 10.655,E2 178.578} C_DIS
Enddeposition()
LIN {X 0.9547,Y -131.6551,Z 168,A -87.8637,B 10.6484,C 0.2927,E1 10.655,E2 178.578} C_DIS
Startdeposition()
$VEL.CP = VEL_PRINT
LIN {X -0.8275,Y -132.5732,Z 168,A -89.0696,B 10.6479,C 0.309,E1 10.6513,E2 179.872} C_DIS
LIN {X -4.8514,Y -132.4872,Z 168,A -90.8855,B 10.6479,C 0.3108,E1 10.6462,E2 181.6979} C_DIS
LIN {X -9.3544,Y -132.2455,Z 168,A -92.8003,B 10.6479,C 0.3099,E1 10.6409,E2 183.6093} C_DIS
LIN {X -13.0214,Y -131.935,Z 168,A -94.3076,B 10.6479,C 0.3079,E1 10.6367,E2 185.1071} C_DIS
LIN {X -16.2756,Y -131.574,Z 168,A -95.8149,B 10.6479,C 0.3096,E1 10.6325,E2 186.6262} C_DIS
LIN {X -20.0631,Y -131.0488,Z 168,A -97.4299,B 10.6479,C 0.3083,E1 10.628,E2 188.2371} C_DIS
LIN {X -23.5658,Y -130.4643,Z 168,A -98.9032,B 10.6479,C 0.3064,E1 10.624,E2 189.7034} C_DIS
LIN {X -27.0376,Y -129.7905,Z 168,A -100.4446,B 10.6479,C 0.306,E1 10.6198,E2 191.2469} C_DIS
LIN {X -30.5629,Y -129.0054,Z 168,A -102.1478,B 10.6479,C 0.3082,E1 10.6151,E2 192.9677} C_DIS
LIN {X -34.2153,Y -128.0841,Z 168,A -103.6574,B 10.648,C 0.3047,E1 10.611,E2 194.4633} C_DIS
LIN {X -37.3838,Y -127.1954,Z 168,A -105.1359,B 10.648,C 0.3049,E1 10.6071,E2 195.9488} C_DIS
LIN {X -41.4611,Y -125.9261,Z 168,A -107.1496,B 10.648,C 0.3071,E1 10.6016,E2 197.9831} C_DIS
LIN {X -45.3694,Y -124.5712,Z 168,A -108.7548,B 10.648,C 0.3017,E1 10.5975,E2 199.5665} C_DIS
LIN {X -48.5112,Y -123.3823,Z 168,A -110.3324,B 10.648,C 0.303,E1 10.5933,E2 201.1594} C_DIS
LIN {X -52.7862,Y -121.6134,Z 168,A -112.1986,B 10.6482,C 0.2981,E1 10.5886,E2 203.0096} C_DIS
LIN {X -55.8783,Y -120.2241,Z 168,A -113.7148,B 10.6482,C 0.2976,E1 10.5847,E2 204.532} C_DIS
LIN {X -58.8151,Y -118.8149,Z 168,A -115.1221,B 10.6482,C 0.2959,E1 10.5812,E2 205.9392} C_DIS
LIN {X -62.2734,Y -117.0414,Z 168,A -116.8211,B 10.6482,C 0.2942,E1 10.577,E2 207.6405} C_DIS
LIN {X -65.3974,Y -115.3256,Z 168,A -118.4769,B 10.6482,C 0.2946,E1 10.5729,E2 209.3101} C_DIS
LIN {X -69.5054,Y -112.897,Z 168,A -120.3361,B 10.6485,C 0.2875,E1 10.5685,E2 211.1445} C_DIS
LIN {X -72.4969,Y -111.0001,Z 168,A -122.0805,B 10.6485,C 0.2896,E1 10.5643,E2 212.9144} C_DIS
LIN {X -76.2569,Y -108.451,Z 168,A -123.9673,B 10.6485,C 0.285,E1 10.56,E2 214.7917} C_DIS
LIN {X -79.2531,Y -106.2809,Z 168,A -125.5996,B 10.6485,C 0.2831,E1 10.5563,E2 216.4276} C_DIS
LIN {X -82.4576,Y -103.8145,Z 168,A -127.3936,B 10.6486,C 0.281,E1 10.5524,E2 218.2268} C_DIS
LIN {X -85.7933,Y -101.0753,Z 168,A -129.3489,B 10.6486,C 0.2795,E1 10.5482,E2 220.1924} C_DIS
LIN {X -88.7404,Y -98.4986,Z 168,A -131.0107,B 10.6488,C 0.2758,E1 10.5447,E2 221.8501} C_DIS
LIN {X -91.8975,Y -95.5599,Z 168,A -132.8629,B 10.6488,C 0.2719,E1 10.541,E2 223.7002} C_DIS
LIN {X -94.9709,Y -92.5061,Z 168,A -134.8172,B 10.6489,C 0.2698,E1 10.5371,E2 225.6635} C_DIS
LIN {X -98.0759,Y -89.2067,Z 168,A -136.7537,B 10.649,C 0.2653,E1 10.5334,E2 227.5966} C_DIS
LIN {X -101.0311,Y -85.8452,Z 168,A -138.6886,B 10.6491,C 0.2612,E1 10.5299,E2 229.5307} C_DIS
LIN {X -104.1024,Y -82.0941,Z 168,A -140.8434,B 10.6492,C 0.2577,E1 10.5261,E2 231.6915} C_DIS
LIN {X -106.8186,Y -78.5269,Z 168,A -142.7444,B 10.6494,C 0.2526,E1 10.5229,E2 233.5872} C_DIS
LIN {X -109.3382,Y -74.979,Z 168,A -144.5575,B 10.6494,C 0.2469,E1 10.52,E2 235.3911} C_DIS
LIN {X -111.6044,Y -71.5622,Z 168,A -146.4481,B 10.6495,C 0.245,E1 10.5171,E2 237.2948} C_DIS
LIN {X -113.671,Y -68.2332,Z 168,A -148.2243,B 10.6495,C 0.2424,E1 10.5145,E2 239.0799} C_DIS
LIN {X -115.7922,Y -64.5676,Z 168,A -149.9441,B 10.6497,C 0.2357,E1 10.5122,E2 240.7853} C_DIS
LIN {X -117.7715,Y -60.8828,Z 168,A -151.7679,B 10.6498,C 0.2315,E1 10.5098,E2 242.6098} C_DIS
LIN {X -120.4983,Y -55.2854,Z 168,A -154.4066,B 10.65,C 0.2235,E1 10.5066,E2 245.2404} C_DIS
LIN {X -121.7245,Y -52.5293,Z 168,A -155.8211,B 10.65,C 0.2222,E1 10.505,E2 246.6671} C_DIS
LIN {X -123.0324,Y -49.3887,Z 168,A -157.3104,B 10.65,C 0.2186,E1 10.5034,E2 248.1576} C_DIS
LIN {X -124.2622,Y -46.208,Z 168,A -158.7927,B 10.6502,C 0.2148,E1 10.502,E2 249.6398} C_DIS
LIN {X -125.376,Y -43.0948,Z 168,A -160.2318,B 10.6502,C 0.2111,E1 10.5006,E2 251.0789} C_DIS
LIN {X -126.5396,Y -39.5546,Z 168,A -161.8784,B 10.6503,C 0.2073,E1 10.4992,E2 252.7286} C_DIS
LIN {X -127.3291,Y -36.9272,Z 168,A -163.0581,B 10.6503,C 0.2039,E1 10.4983,E2 253.9066} C_DIS
LIN {X -129.0676,Y -30.3052,Z 168,A -166.0636,B 10.6505,C 0.1965,E1 10.4962,E2 256.9151} C_DIS
LIN {X -129.7673,Y -27.1519,Z 168,A -168.3332,B 10.6503,C 0.2089,E1 10.4949,E2 259.2863} C_DIS
LIN {X -130.8415,Y -21.3766,Z 168,A -170.0224,B 10.6507,C 0.1857,E1 10.4941,E2 260.8732} C_DIS
LIN {X -131.3054,Y -18.3129,Z 168,A -171.5676,B 10.6507,C 0.1857,E1 10.4935,E2 262.4416} C_DIS
LIN {X -131.8167,Y -14.1647,Z 168,A -173.3044,B 10.6508,C 0.1792,E1 10.4929,E2 264.1685} C_DIS
LIN {X -132.1922,Y -10.0846,Z 168,A -175.1212,B 10.6508,C 0.1749,E1 10.4925,E2 265.989} C_DIS
LIN {X -132.4383,Y -6.062,Z 168,A -176.9794,B 10.6509,C 0.172,E1 10.4922,E2 267.8593} C_DIS
LIN {X -132.561,Y -1.9893,Z 168,A -178.6127,B 10.6511,C 0.1644,E1 10.4922,E2 269.4757} C_DIS
LIN {X -132.555,Y 2.3464,Z 168,A 179.4889,B 10.6511,C 0.1594,E1 10.4922,E2 271.3751} C_DIS
LIN {X -132.4473,Y 5.8754,Z 168,A 177.9332,B 10.6511,C 0.1555,E1 10.4923,E2 272.9329} C_DIS
LIN {X -132.2329,Y 9.5268,Z 168,A 176.3305,B 10.6513,C 0.1513,E1 10.4926,E2 274.5364} C_DIS
LIN {X -131.946,Y 12.9073,Z 168,A 174.7546,B 10.6513,C 0.149,E1 10.493,E2 276.1236} C_DIS
LIN {X -131.1549,Y 19.3656,Z 168,A 171.2942,B 10.6513,C 0.1529,E1 10.4944,E2 279.6569} C_DIS
LIN {X -130.2935,Y 24.495,Z 168,A 169.6946,B 10.6515,C 0.1344,E1 10.4951,E2 281.1784} C_DIS
LIN {X -129.0233,Y 30.4888,Z 168,A 167.1252,B 10.6515,C 0.1253,E1 10.4966,E2 283.7358} C_DIS
Enddeposition()
END
